		IF conveyorPos >= currentBundle.length AND NOT occupied THEN //rear of bundle has cleared the area
			status := SectionTask.COMPLETE;
		END_IF
		
	SectionTask.COMPLETE:	
		iBundle := iBundle + 1;
		//bundleOut := GVL.nullBundle;
		MEMSET(ADR(activeBundle), 0, SIZEOF(activeBundle));
		
		status := SectionTask.IDLE;
		
		runSectionTasks := TRUE;
		
	-100: //previously completed bundle reversed into this section		
		pConveyorMode := ConveyorMode.FORWARD;
		
		IF NOT occupied AND conveyorPos = 0 THEN
			status := SectionTask.ALIGN;
		END_IF
		
END_CASE
END_METHOD

METHOD shiftIterator : BOOL
//2023-10-24 - array of pointers replaced with iterator for MAIN's queue passed by pointer
iBundle := iBundle - 1;
END_METHOD

METHOD PROTECTED ABSTRACT unload : BOOL
VAR_INPUT
END_VAR
(*
unload, unstage, etc
*)
END_METHOD

END_FUNCTION_BLOCK

// ---- DUTs/Hardware/Conveyors/ConveyorSC.TcPOU
FUNCTION_BLOCK ConveyorSC
VAR_INPUT
	bEnable : BOOL;
END_VAR
VAR_OUTPUT
	trueMode : ConveyorMode;
	requestedMode : ConveyorMode;
	
	error AT %I* : BOOL;
	position AT %I* : REAL;
	velocity AT %I* : REAL;
END_VAR
VAR
	enable AT %Q* : BOOL := TRUE;
	direction AT %Q* : BOOL; //FALSE = forward, TRUE = backward
	pulse AT %Q* : BOOL;
	reset AT %Q* : BOOL;
	
	sensorEntry AT %I* : BOOL := TRUE;
	sensorExit AT %I* : BOOL;
END_VAR
VAR
	//nextConveyor : POINTER TO ConveyorSC;
	//prevConveyor : POINTER TO ConveyorSC;
	
	pulser : TP; //pulses are assumed to be low-high-low
END_VAR
VAR_STAT CONSTANT
	pulseWidth : TIME := T#50MS;
END_VAR
(*
standard slat conveyor - no lifter
compliant with PLCopen motion control
*)

enable := bEnable;

override();

sequence();

METHOD backward : BOOL
VAR_INPUT
END_VAR
END_METHOD

METHOD forward : BOOL
VAR_INPUT
END_VAR
END_METHOD

{attribute 'monitoring' := 'call'}
PROPERTY IsOccupied : BOOL
GET
IsOccupied := sensorExit OR sensorEntry;
END_GET
END_PROPERTY

METHOD join : BOOL
VAR_INPUT
	conveyor : POINTER TO ConveyorSC;
END_VAR
//nextConveyor := conveyor;
//conveyor^.prevConveyor := THIS;
END_METHOD

METHOD PROTECTED override : BOOL
VAR_INPUT
END_VAR
END_METHOD

METHOD reset : BOOL
VAR_INPUT
END_VAR
position := 0;
velocity := velocity; //no change
END_METHOD

METHOD PROTECTED sequence : BOOL
VAR_INPUT
END_VAR
direction := (trueMode = ConveyorMode.BACKWARD); //set direction bit

pulser(IN:= , PT:= pulseWidth, Q=> pulse, ET=> );
pulser.IN := 
	enable AND 
	NOT error AND 
	NOT reset AND 
	(trueMode = ConveyorMode.FORWARD OR trueMode = ConveyorMode.BACKWARD)
	AND pulser.Q; //ends pulse itself
END_METHOD

METHOD setMode : BOOL
VAR_INPUT
	mode : ConveyorMode;
END_VAR
trueMode := mode;
END_METHOD

METHOD setRequest : BOOL
VAR_INPUT
	newRequest : ConveyorMode;
END_VAR
requestedMode := newRequest;
END_METHOD

METHOD target : BOOL
VAR_INPUT
	targetPosition : REAL;
END_VAR
END_METHOD

END_FUNCTION_BLOCK

// ---- DUTs/Hardware/Conveyors/Conveyor.TcPOU
FUNCTION_BLOCK Conveyor
VAR_INPUT
	bEnable : BOOL;
END_VAR
VAR_OUTPUT	
	enable AT %Q* : BOOL;
	direction AT %Q* : BOOL; //FALSE = forward, TRUE = backward
	pulse AT %Q* : BOOL;
	reset AT %Q* : BOOL;
	
	error AT %I* : BOOL;
	sensorEntry AT %I* : BOOL;
	sensorExit AT %I* : BOOL;
	
	//vertical conveyors only
	requestLifter: BOOL;

	lifterEnable AT %Q* : BOOL := TRUE;
	lifterDirection AT %Q* : BOOL; //FALSE = up, TRUE = down
	lifterPulse AT %Q* : BOOL;
	lifterReset AT %Q* : BOOL;
	
	lifterError AT %I* : BOOL;
	extended AT %I* : BOOL;
	retracted AT %I* : BOOL;
END_VAR
VAR_OUTPUT
	position AT %I* : REAL;
	velocity AT %I* : REAL;
END_VAR
VAR
	operation : ConveyorMode;
	request : ConveyorMode;
	
	//pulses are assumed to be low-HIGH-low
	pulser : TP;
	lifterPulser : TP;
	
	hasLifter : BOOL;
END_VAR
VAR_STAT CONSTANT
	pulseWidth : TIME := T#25MS;
END_VAR

pulser(IN:= , PT:= pulseWidth, Q=> pulse, ET=> );

direction := (operation = ConveyorMode.BACKWARD);

pulser.IN := 
	enable AND 
	NOT error AND 
	NOT reset AND 
	(operation = ConveyorMode.FORWARD OR operation = ConveyorMode.BACKWARD);

IF pulser.IN AND NOT pulser.Q THEN
	pulser.IN := FALSE;
END_IF

lifterPulser(IN:= , PT:= pulseWidth, Q=> lifterPulse, ET=> );

lifterPulser.IN := 
	hasLifter AND
	lifterEnable AND 
	NOT lifterError AND 
	NOT lifterReset AND 
	requestLifter;
	
IF lifterPulser.IN AND NOT lifterPulser.Q THEN
	lifterPulser.IN := FALSE;
END_IF

METHOD backward : BOOL
VAR_INPUT
END_VAR
END_METHOD

METHOD extend : BOOL
VAR_INPUT
END_VAR
END_METHOD

METHOD forward : BOOL
VAR_INPUT
END_VAR
END_METHOD

{attribute 'monitoring' := 'call'}
PROPERTY IsOccupied : BOOL
GET
IsOccupied := sensorExit OR sensorEntry;
END_GET
END_PROPERTY

METHOD reset : BOOL
VAR_INPUT
END_VAR
position := 0;
velocity := velocity; //no change

extend();
END_METHOD

METHOD retract : BOOL
VAR_INPUT
END_VAR
END_METHOD

METHOD setOperation : BOOL
VAR_INPUT
	newOperation : ConveyorMode;
END_VAR
operation := newOperation;
END_METHOD

METHOD setRequest : BOOL
VAR_INPUT
	newRequest : ConveyorMode;
END_VAR
request := newRequest;
END_METHOD

METHOD target : BOOL
VAR_INPUT
	targetPosition : REAL;
END_VAR
END_METHOD

END_FUNCTION_BLOCK

// ---- DUTs/Hardware/Robots/RobotA22.TcPOU
FUNCTION_BLOCK RobotA22 EXTENDS KukaRobot
VAR_INPUT
	wrapSafety : BOOL;
END_VAR
VAR_OUTPUT //from outputs array
	taskID : TaskA22;
	param1 : INT;
	param2 : INT;
	Xmm : INT;
	Ymm : INT;
	Zmm : INT;
	angle : INT;
	foldPosition0 : INT;
	foldPosition1 : INT;
END_VAR
VAR_OUTPUT //from inputs array
	tool : SectionEnum := SectionEnum.CARDBOARD_CORNERGUARD;
	suspendedMaterial : STRING;
	
	completedTask : TaskA22;
	eoatDistance : INT;
	cardboardAvailability : INT;
	cornerGuardAvailability : INT;
	materialAtHoldingPosition : INT;
	//grp6
	//grp7
	
	wrapSafetyIn : BOOL;
	
END_VAR
VAR //HMI data
	reservationEnum : SectionEnum;
	hmiTask : STRING;
	hmiTool : STRING;
END_VAR

{warning disable C0195}
SUPER^();

outputs[1] := taskID;
outputs[2] := param1;
outputs[3] := param2;
outputs[4] := Xmm;
outputs[5] := Ymm;
outputs[6] := Zmm;
outputs[7] := angle;
outputs[8] := foldPosition0;
outputs[9] := foldPosition1;

refreshParameters();

reservationEnum := reservation;
IF reservationEnum = SectionEnum.NULL_SECTION THEN
	hmiReservation := 'N/A';
ELSE
	hmiReservation := TO_STRING(reservationEnum);
END_IF

hmiTask := TO_STRING(taskID);
hmiTool := TO_STRING(tool);

{attribute 'monitoring' := 'call'}
PROPERTY Busy : BOOL
GET
VAR
	//emptyOutput : ARRAY[1..50] OF INT;
END_VAR
//Busy stays TRUE until outputs are cleared AND completed task has elapsed
//Ready is always inverse of Busy
refreshParameters();

Busy := taskID <> 0 OR completedTask <> 0;
END_GET
END_PROPERTY

METHOD changeEOAT : BOOL
VAR_INPUT
	targetTool : SectionEnum;
END_VAR
//fill in IO here

changeEOAT := TRUE;
END_METHOD

METHOD clearCommand : BOOL
VAR_INPUT
END_VAR
SUPER^.clearCommand();

refreshParameters();
END_METHOD

{attribute 'monitoring' := 'call'}
PROPERTY Done : BOOL
GET
refreshParameters();

Done :=
	completedTask = taskID AND
	taskID <> 0 AND
	completedTask <> 0;
END_GET
END_PROPERTY

{attribute 'monitoring' := 'call'}
PROPERTY HoldMaterial : STRING
GET
HoldMaterial := suspendedMaterial;
END_GET
SET
suspendedMaterial := HoldMaterial;
END_SET
END_PROPERTY

{attribute 'monitoring' := 'call'}
PROPERTY Ready : BOOL
GET
refreshParameters();

Ready := taskID = 0 AND completedTask = 0;
END_GET
END_PROPERTY

METHOD PRIVATE refreshParameters : BOOL
VAR_INPUT
END_VAR
{warning disable C0196}
taskID := outputs[1];
param1 := outputs[2];
param2 := outputs[3];
Xmm := outputs[4];
Ymm := outputs[5];
Zmm := outputs[6];
angle := outputs[7];
foldPosition0 := outputs[8];
foldPosition1 := outputs[9];

completedTask := inputs[1];
(*
eoatDistance := inputs[2];
magazineAvailability := inputs[3];
chipboardSkidInPosition := inputs[4];
materialAtHoldingPosition := inputs[5];
//robotEOAT := inputs[6];

strapSafetyIn := inputs[4].15;
*)
END_METHOD

METHOD setGroup : BOOL
VAR_INPUT
	group : INT;
	value : INT;
END_VAR
SUPER^.setGroup(group := group, value := value);

refreshParameters();
END_METHOD

METHOD setParameters : BOOL
VAR_INPUT
	newTaskID : INT;
	newParam1 : INT;
	newParam2 : INT;
	newXmm : INT;
	newYmm : INT;
	newZmm : INT;
	newAngle : INT;
	newStagingOccupancy : INT;
	newInsertionSuctionStatus : INT;
	newMagazineStatus : INT; //unused
	newInspectionValue : INT;
END_VAR
setGroup(group := 1, value := newTaskID);
setGroup(group := 2, value := newParam1);
setGroup(group := 3, value := newParam2);
setGroup(group := 4, value := newXmm);
setGroup(group := 5, value := newYmm);
setGroup(group := 6, value := newZmm);
setGroup(group := 7, value := newAngle);

newStagingOccupancy.15 := wrapSafety;
setGroup(group := 8, value := newStagingOccupancy);

setGroup(group := 9, value := newInsertionSuctionStatus);
setGroup(group := 10, value := newMagazineStatus);
setGroup(group := 11, value := newInspectionValue);

refreshParameters();
END_METHOD

END_FUNCTION_BLOCK

// ---- DUTs/Hardware/Material Holders/SkidMagazine.TcPOU
FUNCTION_BLOCK SkidMagazine EXTENDS MaterialHolder
VAR_OUTPUT
	inPosition AT %I* : ARRAY[1..2] OF BOOL;
END_VAR

SUPER^();

METHOD setOccupancy : BOOL
VAR_INPUT
	i : INT;
	occupancy : BOOL;
END_VAR
VAR_OUTPUT
	errorBounds : BOOL;
END_VAR
errorBounds := i < LOWER_BOUND(slots, 1) OR i > UPPER_BOUND(slots, 1);

IF NOT errorBounds THEN
	slots[i].occupied := occupancy;
END_IF
END_METHOD

END_FUNCTION_BLOCK

// ---- DUTs/Hardware/Insertion Package/Insertion.TcPOU
FUNCTION_BLOCK Insertion //2d insertion that combines a slider (alignment) and screw (push)
VAR_INPUT //interface references to existing drives
	slider : I_PositionalDrive;
	screw : I_ContinuousDrive;
END_VAR
VAR_OUTPUT
	contact AT %I* : BOOL;
	
	active : BOOL;
	error : BOOL;
	home : BOOL;
	
	homingComplete : BOOL;
	
	sliderPos : LREAL;
END_VAR
(*
this FB encapsulates 2 drives into a generic insertion machine
both drives should be declared externally in Hardware GVL as a concrete FB
Insertion instance should be declared and called in module scope, with the drives from Hardware GVL passed in by Interface reference
*)

homingComplete := slider.HomeSet AND screw.HomeSet;

active := slider.Active OR screw.Active;
error := slider.Error OR screw.Error;
home := slider.AtHome AND screw.AtHome;

sliderPos := slider.CurrentPosition;

METHOD align : BOOL
VAR_INPUT
	targetPos : REAL;
END_VAR
slider.moveAbsolute(newTarget := targetPos);
END_METHOD

METHOD homingSequence : BOOL
VAR_INPUT
END_VAR
IF NOT slider.homeSet THEN
	slider.homingSequence();
END_IF

IF NOT screw.homeSet THEN
	screw.homingSequence();
END_IF

homingSequence := homingComplete;
END_METHOD

METHOD press : BOOL
VAR_INPUT
END_VAR
IF NOT contact THEN
	screw.moveContinuous(direction := MC_Negative_Direction);
END_IF
END_METHOD

METHOD release : BOOL
VAR_INPUT
END_VAR
screw.moveContinuous(direction := MC_Positive_Direction);
END_METHOD

METHOD reset : BOOL
VAR_INPUT
END_VAR
slider.reset();
screw.reset();
END_METHOD

METHOD stop : BOOL
VAR_INPUT
END_VAR
screw.stop();
slider.stop();
END_METHOD

METHOD toHome : BOOL
VAR_INPUT
END_VAR
slider.toHome();
screw.toHome();

toHome := slider.AtHome AND screw.AtHome;
END_METHOD

END_FUNCTION_BLOCK

// ---- POUs/Helper Functions/Material Functions/MatchesMaterialType.TcPOU
FUNCTION MatchesMaterialType : BOOL
VAR_INPUT
	pair : REFERENCE TO PositionMaterials;
	materialPrefix : STRING;
END_VAR
VAR
END_VAR

MatchesMaterialType :=
	FIND(pair.top, materialPrefix) > 0 AND
	FIND(pair.left, materialPrefix) > 0 AND
	FIND(pair.right, materialPrefix) > 0 AND
	FIND(pair.bottom, materialPrefix) > 0 AND
	
	FIND(pair.topLeft, materialPrefix) > 0 AND
	FIND(pair.topRight, materialPrefix) > 0 AND
	FIND(pair.bottomLeft, materialPrefix) > 0 AND
	FIND(pair.bottomRight, materialPrefix) > 0 ;

END_FUNCTION

// ---- Sections/A21a - Chipboard/ChipboardEx.TcPOU
FUNCTION_BLOCK ChipboardEx EXTENDS SectionEx
VAR_IN_OUT
	A21_SC_C18 : ConveyorSC;
	A21_LSC_C19 : ConveyorLSC;
	A21_LSC_C20 : ConveyorLSC;
END_VAR
VAR_IN_OUT
	robotLeft, robotRight : RobotA21;
	toolStorageLeft, toolStorageRight : A21ToolStorage;
	
	skidLeft, skidRight : SkidMagazine;
END_VAR
VAR	
	step : (IDLE, RETRACT_CONVEYOR, LOAD_CIP, EXTEND_CONVEYOR, COMPLETE := 1050);
	
	loadSet : INT;
END_VAR
VAR //bundle data
	materialsArr : (*REFERENCE TO*) ARRAY[0..CONSTS.maxPairs] OF PositionMaterials;
END_VAR
VAR
	aoiLoadLeft, aoiLoadRight : AOI_LoadChipboard;
	
	pushSmallConveyorPos : REAL;
	pushLargeConveyorPos : REAL;
END_VAR

aoiBlocks(); //call AOIs and large library FBs

SUPER^();

METHOD PROTECTED aoiBlocks : BOOL
VAR_INPUT
END_VAR
{warning disable C0371}
aoiLoadRight(
	sectionID:= sectionID, 
	execute:= ,
	robot:= robotRight, 
	storage:= skidRight,
	loadedMaterials:= loadedMaterials,
	surfaceID:= , 
	material:= , 
	loadedMaterials=> , 
	done=> , 
	error=> );
	
aoiLoadRight(
	sectionID:= sectionID, 
	execute:= , 
	robot:= robotRight, 
	storage:= skidRight,
	loadedMaterials:= loadedMaterials, 
	surfaceID:= , 
	material:= , 
	busy=> , 
	done=> , 
	error=> , 
	recovery=> , 
	failCounter=> );
END_METHOD

METHOD PROTECTED load : BOOL
VAR_INPUT
	pairIndex : INT;
END_VAR
VAR_OUTPUT
	error : BOOL;
END_VAR
VAR
	pair : REFERENCE TO PositionMaterials REF= materialsArr[pairIndex];
END_VAR
{warning disable C0371}
IF robotLeft.error AND robotLeft.error THEN
	error := TRUE;
	RETURN;

ELSIF
	( robotLeft.reservation <> sectionID AND_THEN robotLeft.reserve(sectionID) ) OR
	( robotRight.reservation <> sectionID AND_THEN robotRight.reserve(sectionID) ) THEN
	RETURN;
	
ELSIF //wrong tool and not finished changing tool
	(robotLeft.tool <> sectionID AND_THEN NOT robotLeft.changeEOAT(targetTool := sectionID)) OR
	(robotRight.tool <> sectionID AND_THEN NOT robotRight.changeEOAT(targetTool := sectionID))
THEN
	RETURN;
END_IF
//robots ok

CASE loadSet OF
	0: //left robot -> top, right robot -> bottom
		IF aoiLoadLeft.done AND aoiLoadRight.done THEN
			aoiLoadLeft.execute := aoiLoadRight.execute := FALSE;
			loadSet := 10;
			RETURN;
		END_IF
		
		aoiLoadLeft.surfaceID := Surface.TOP;
		aoiLoadLeft.material := pair.left;
		
		aoiLoadRight.surfaceID := Surface.BOTTOM;
		aoiLoadRight.material := pair.right;
		
		aoiLoadLeft.execute := NOT aoiLoadLeft.recovery;
		aoiLoadRight.execute := NOT aoiLoadRight.recovery;
		
	10: //recovery		
		IF robotRight.error THEN //left ok, right error
			
			IF aoiLoadLeft.done THEN
				aoiLoadLeft.execute := FALSE;
				loadSet := COMPLETE;
				RETURN;
			END_IF
			
			aoiLoadLeft.surfaceID := Surface.BOTTOM;
			aoiLoadLeft.material := pair.bottom;
			aoiLoadLeft.execute := NOT aoiLoadLeft.recovery;
			
		ELSIF robotLeft.error THEN //left error, right ok
			
			IF aoiLoadRight.done THEN
				aoiLoadRight.execute := FALSE;
				loadSet := COMPLETE;
				RETURN;
			END_IF
			
			aoiLoadRight.surfaceID := Surface.TOP;
			aoiLoadRight.material := pair.top;
			aoiLoadRight.execute := NOT aoiLoadRight.recovery;
			
		END_IF
		
	COMPLETE:
		loadSet := 0;
		
		robotLeft.release(sectionID);
		robotRight.release(sectionID);
		
		load := TRUE;
END_CASE
END_METHOD

METHOD PRIVATE loadingSequence : BOOL
VAR_IN_OUT
	robot : RobotA21;
	storage : SkidMagazine;
	loadStep : INT;
END_VAR
VAR_INPUT
	surfaceID : Surface;
	material : STRING;
END_VAR
VAR_OUTPUT
	fail : BOOL;
END_VAR
VAR
	slot : INT;
END_VAR
VAR CONSTANT
	suctionDistance : INT := 10;
END_VAR
{warning disable C0371}
IF material = '' THEN
	loadingSequence := TRUE;
	RETURN;
END_IF

CASE loadStep OF
	0:
		robot.clearCommand();
		IF robot.Ready THEN
			loadStep := 1;
		END_IF
	
	1:
		IF surfaceID = Surface.BOTTOM (*AND_THEN conveyors not retracted*) THEN
			//retract conveyors
			RETURN;
		END_IF
		loadStep := 10;
		
	10: //grab from chipboard skid
		IF NOT storage.findSlot(material := material, index => slot) THEN
			fail := TRUE;
			RETURN;
		(*
		ELSIF surfaceID = Surface.BOTTOM (*AND_THEN (*conveyor not lowered*)*) THEN
			//lower conveyor
			RETURN;
		*)
		END_IF
		
		IF robot.eoatDistance < suctionDistance THEN
			robot.HoldMaterial := storage.getSlot(i := slot);
		END_IF
		
		IF robot.Done THEN
			loadStep := COMPLETE;
			RETURN;
		ELSIF robot.materialAtHoldingPosition.4 OR robot.materialAtHoldingPosition.5 THEN //bits 4 and 5 are chipboard in position
			loadStep := 20;
			RETURN;
		END_IF
		
		robot.setGroup(group := 1, value := TaskA21.PLACE_CHIPBOARD_TOP);
		robot.setGroup(group := 2, value := slot);
		
	20: //place to bundle
		IF robotLeft.Done THEN
			loadStep := COMPLETE;
			RETURN;
		END_IF
		
		IF robot.HoldMaterial <> '' THEN
			loadedMaterials[surfaceID] := robot.HoldMaterial;
			robot.HoldMaterial := '';
		END_IF
		
	COMPLETE:
		IF loadedMaterials[surfaceID] = material THEN
			loadingSequence := TRUE;
		ELSE
			loadStep := 0;
		END_IF
		
END_CASE
END_METHOD

METHOD PROTECTED maintenance : BOOL
VAR_INPUT
END_VAR
{warning disable C0371}
//no specific tasks yet, free run and testing

IF robotLeft.Done THEN
	robotLeft.clearCommand();
END_IF

IF robotRight.Done THEN
	robotRight.clearCommand();
END_IF
END_METHOD

METHOD PROTECTED manual : BOOL
VAR_INPUT
END_VAR
END_METHOD

METHOD PROTECTED process : BOOL
VAR_INPUT
	auto : BOOL;
END_VAR
VAR_OUTPUT
	error : BOOL;
END_VAR
CASE step OF
	IDLE:
		IF trigger.Q THEN
			step := RETRACT_CONVEYOR;
		END_IF
		
	RETRACT_CONVEYOR:
		(*
		IF demoPair.bottom <> '' (*retract conveyors*) THEN
			IF TRUE (*BLSC 1-3 retracted*) THEN
				done := TRUE;
			END_IF
		ELSE
			done := TRUE;
		END_IF
		
		IF
			(manualStep AND_THEN execute) OR
			(NOT manualStep AND_THEN done)
		THEN
			done := FALSE;
			step := LOAD_MATERIAL;
		END_IF
		*)
		step := LOAD_CIP;
	LOAD_CIP:
		IF NOT done THEN
			done := load(pairIndex:= iPair, error=> error);
		END_IF
		
		IF
			(auto AND done) OR
			(NOT auto AND_THEN trigger.Q)
		THEN
			done := FALSE;
			
			step := EXTEND_CONVEYOR;
		END_IF
		
	EXTEND_CONVEYOR:
		(*
		IF FALSE (*conveyors not extended*) THEN
			//extend conveyors
		END_IF
		
		IF
			(auto AND done) OR
			(NOT auto AND_THEN execute) //conveyors extended
		THEN
			done := FALSE;
			step := COMPLETE;
		END_IF
		*)
		step := COMPLETE;
	COMPLETE:
		//reset everything
		step := IDLE;
		
		process := TRUE;
		
END_CASE
END_METHOD

METHOD PROTECTED ps_AbortCondition : BOOL
VAR_INPUT
END_VAR
{warning disable C0371}
ps_AbortCondition :=
	robotLeft.error OR 
	robotRight.error;
END_METHOD

METHOD PROTECTED ps_Aborted : BOOL
VAR_INPUT
END_VAR
ps_Aborted := TRUE;
END_METHOD

METHOD PROTECTED ps_Aborting : BOOL
VAR_INPUT
END_VAR
{warning disable C0371}
aoiLoadLeft.reset();
aoiLoadRight.reset();

robotLeft.clearCommand();
robotRight.clearCommand();

//stop conveyors

ps_Aborting :=
	NOT robotLeft.Busy AND
	NOT robotRight.Busy;
END_METHOD

METHOD PROTECTED ps_Clearing : BOOL
VAR_INPUT
END_VAR
{warning disable C0371}
(*reset conveyors*)

ps_Clearing := 
	NOT robotLeft.error AND
	NOT robotRight.error;
END_METHOD

METHOD PROTECTED ps_Complete : BOOL
VAR_INPUT
END_VAR
ps_Complete := TRUE;
END_METHOD

METHOD PROTECTED ps_Completing : BOOL
VAR_INPUT
END_VAR
ps_Completing := NOT occupied;
END_METHOD

METHOD PROTECTED ps_Held : BOOL
VAR_INPUT
END_VAR
ps_Held := NOT hold;
END_METHOD

METHOD PROTECTED ps_HoldCondition : BOOL
VAR_INPUT
END_VAR
END_METHOD

METHOD PROTECTED ps_Holding : BOOL
VAR_INPUT
END_VAR
{warning disable C0371}
//set robot to pause

ps_Holding := TRUE;
END_METHOD

METHOD PROTECTED ps_Resetting : BOOL
VAR_INPUT
END_VAR
{warning disable C0371}
(*reset conveyors*)

ps_Resetting := 
	reset AND
	NOT robotLeft.error AND
	NOT robotRight.error;
END_METHOD

METHOD PROTECTED ps_Starting : BOOL
VAR_INPUT
END_VAR
{warning disable C0371}
//extend conveyors

ps_Starting := TRUE; //conveyors extended
END_METHOD

METHOD PROTECTED ps_StopCondition : BOOL
VAR_INPUT
END_VAR
ps_StopCondition := 
	stop;
END_METHOD

METHOD PROTECTED ps_Stopped : BOOL
VAR_INPUT
END_VAR
ps_Stopped := TRUE;
END_METHOD

METHOD PROTECTED ps_Stopping : BOOL
VAR_INPUT
END_VAR
{warning disable C0371}
aoiLoadLeft.reset();
aoiLoadRight.reset();

robotLeft.clearCommand();
robotRight.clearCommand();

//stop conveyors

ps_Stopping :=
	NOT robotLeft.Busy AND
	NOT robotRight.Busy;
END_METHOD

METHOD PROTECTED ps_SuspendCondition : BOOL
VAR_INPUT
END_VAR
END_METHOD

METHOD PROTECTED ps_Suspended : BOOL
VAR_INPUT
END_VAR
ps_Suspended := NOT ps_SuspendCondition();
END_METHOD

METHOD PROTECTED ps_Suspending : BOOL
VAR_INPUT
END_VAR
ps_Suspending := TRUE;
END_METHOD

METHOD PROTECTED ps_Unholding : BOOL
VAR_INPUT
END_VAR
ps_Unholding := TRUE;
END_METHOD

METHOD PROTECTED ps_Unsuspending : BOOL
VAR_INPUT
END_VAR
ps_Unsuspending := TRUE;
END_METHOD

METHOD PROTECTED runSectionTasks : BOOL
VAR_INPUT
	auto : BOOL;
END_VAR
VAR_OUTPUT
	error : BOOL;
END_VAR
SUPER^.runSectionTasks(auto := auto, error => error);

CASE status OF //add additional instructions for each state
	SectionTask.IDLE:
		//
	
	SectionTask.ALIGN:
		//
		
	SectionTask.ACTIVE:
		//
		
	SectionTask.DISCHARGE:
		aoiLoadLeft.reset();
		aoiLoadRight.reset();
		
	SectionTask.COMPLETE:	
		//
		
	-100:
		RETURN;
		
END_CASE
END_METHOD

METHOD PROTECTED unload : BOOL
VAR_INPUT
END_VAR
//unload from insertion
//remove from staging table
END_METHOD

END_FUNCTION_BLOCK

// ---- DUTs/Hardware/Robots/RobotA21.TcPOU
FUNCTION_BLOCK RobotA21 EXTENDS KukaRobot
VAR_INPUT
	strapSafety : BOOL;
END_VAR
VAR_OUTPUT //from outputs array
	{warning disable C0195}
	taskID : TaskA21;
	param1 : INT;
	param2 : INT;
	Xmm : INT;
	Ymm : INT;
	Zmm : INT;
	angle : INT;
	stagingOccupancy : INT;
	insertionSuctionStatus : INT;
	magazineStatus : INT; //unused
	inspectionValue : INT;
	
	strapSafetyOut : BOOL;
END_VAR
VAR_OUTPUT //from inputs array
	tool : SectionEnum := SectionEnum.WOOD_BUNK;
	suspendedMaterial : STRING;
	
	completedTask : TaskA21;
	eoatDistance : INT;
	woodBunkAvailability : INT;
	chipboardAvailability : INT;
	materialAtHoldingPosition : INT;
	
	strapSafetyIn : BOOL;
END_VAR
VAR
	reservationEnum : SectionEnum;
	hmiTask : STRING;
	hmiTool : STRING;
END_VAR
(*
extends KukaRobot
	assigns descriptive labels to each IO group from the array
	additional section-specific methods to get/set IO groups
*)

(*
parameters - aliases to IO elements
command - full IO array
*)
{warning disable C0195}
SUPER^();

outputs[1] := taskID;
outputs[2] := param1;
outputs[3] := param2;
outputs[4] := Xmm;
outputs[5] := Ymm;
outputs[6] := Zmm;
outputs[7] := angle;
outputs[8] := stagingOccupancy;
outputs[9] := insertionSuctionStatus;
outputs[10] := magazineStatus;
outputs[11] := inspectionValue;

outputs[8].15 := strapSafety;

refreshParameters();

reservationEnum := reservation;
IF reservationEnum = SectionEnum.NULL_SECTION THEN
	hmiReservation := 'N/A';
ELSE
	hmiReservation := TO_STRING(reservationEnum);
END_IF

hmiTask := TO_STRING(taskID);
hmiTool := TO_STRING(tool);

{attribute 'monitoring' := 'call'}
PROPERTY Busy : BOOL
GET
VAR
	//emptyOutput : ARRAY[1..50] OF INT;
END_VAR
//Busy stays TRUE until outputs are cleared AND completed task has elapsed
//Ready is always inverse of Busy
refreshParameters();

Busy := taskID <> 0 OR completedTask <> 0;
END_GET
END_PROPERTY

METHOD changeEOAT : BOOL
VAR_INPUT
	targetTool : SectionEnum;
END_VAR
setGroup(group := 1, value := TaskA21.TOOL_CHANGE_CHIPBOARD);
setGroup(group := 1, value := TaskA21.TOOL_CHANGE_BUNK);

changeEOAT := tool = targetTool;
END_METHOD

METHOD clearCommand : BOOL
VAR_INPUT
END_VAR
SUPER^.clearCommand();

refreshParameters();
END_METHOD

{attribute 'monitoring' := 'call'}
PROPERTY Done : BOOL
GET
refreshParameters();

Done :=
	completedTask = taskID AND
	taskID <> 0 AND
	completedTask <> 0;
END_GET
END_PROPERTY

{attribute 'monitoring' := 'call'}
PROPERTY HoldMaterial : STRING
GET
HoldMaterial := suspendedMaterial;
END_GET
SET
suspendedMaterial := HoldMaterial;
END_SET
END_PROPERTY

{attribute 'monitoring' := 'call'}
PROPERTY Ready : BOOL
GET
refreshParameters();

Ready := taskID = 0 AND completedTask = 0;
END_GET
END_PROPERTY

METHOD PRIVATE refreshParameters : BOOL
VAR_INPUT
END_VAR
{warning disable C0196}
taskID := outputs[1];
param1 := outputs[2];
param2 := outputs[3];
Xmm := outputs[4];
Ymm := outputs[5];
Zmm := outputs[6];
angle := outputs[7];
stagingOccupancy := outputs[8];
insertionSuctionStatus := outputs[9];
magazineStatus := outputs[10]; //unused
inspectionValue := outputs[11];

completedTask := inputs[1];
eoatDistance := inputs[2];
woodBunkAvailability := inputs[3];
chipboardAvailability := inputs[4];
materialAtHoldingPosition := inputs[5];
//robotEOAT := inputs[6];

strapSafetyIn := inputs[4].15;
END_METHOD

METHOD setGroup : BOOL
VAR_INPUT
	group : INT;
	value : INT;
END_VAR
SUPER^.setGroup(group := group, value := value);

refreshParameters();
END_METHOD

METHOD setParameters : BOOL
VAR_INPUT
	newTaskID : INT;
	newParam1 : INT;
	newParam2 : INT;
	newXmm : INT;
	newYmm : INT;
	newZmm : INT;
	newAngle : INT;
	newStagingOccupancy : INT;
	newInsertionSuctionStatus : INT;
	newMagazineStatus : INT; //unused
	newInspectionValue : INT;
END_VAR
VAR_INPUT
	strapSafety : BOOL;
END_VAR
setGroup(group := 1, value := newTaskID);
setGroup(group := 2, value := newParam1);
setGroup(group := 3, value := newParam2);
setGroup(group := 4, value := newXmm);
setGroup(group := 5, value := newYmm);
setGroup(group := 6, value := newZmm);
setGroup(group := 7, value := newAngle);

newStagingOccupancy.15 := strapSafety;
setGroup(group := 8, value := newStagingOccupancy);

setGroup(group := 9, value := newInsertionSuctionStatus);
setGroup(group := 10, value := newMagazineStatus);
setGroup(group := 11, value := newInspectionValue);

refreshParameters();
END_METHOD

END_FUNCTION_BLOCK

// ---- Sections/A21b - Wood Bunk/WoodBunkEx.TcPOU
FUNCTION_BLOCK WoodBunkEx EXTENDS SectionEx
VAR_IN_OUT
	A21_LSC_C21 : ConveyorLSC;
END_VAR
VAR_IN_OUT
	robotLeft, robotRight : RobotA21;
	toolStorageLeft, toolStorageRight : A21ToolStorage;
	
	stagingTableLeft, stagingTableRight : StagingTable;
	magazineLeft, magazineRight : SkidMagazine;
	
	strapper : StrapMachine;
	
	insertionLeft, insertionRight : Insertion;
	pistonBottom : SimplePiston;
	
	suctionTop : ARRAY[*] OF SuctionPad; (*1..3*)
	suctionLeft : ARRAY[*] OF SuctionPad; (*1..4*)
	suctionRight : ARRAY[*] OF SuctionPad; (*1..4*)
	suctionBottom : ARRAY[*] OF SuctionPad; (*1..2*)
END_VAR
VAR
	step : (IDLE, STAGING, LOAD_WB, PUSH, STRAP, RELEASE, COMPLETE := 1050);
	
	stageStepLeft, stageStepRight : INT;
	loadStepLeft, loadStepRight : INT;
END_VAR
VAR //bundle data
	demoHeight : REAL := 640; //mm
	materialsArr : (*REFERENCE TO*) ARRAY[0..CONSTS.maxPairs] OF PositionMaterials;
END_VAR
VAR
	//AOIs encapsulate functionality and reduce the number of module variables
	aoiTemplateLeft, aoiTemplateRight : AOI_StagingTemplate;
	aoiStageLeft, aoiStageRight : AOI_StageWoodBunk; 
	aoiLoadLeft, aoiLoadRight : AOI_LoadWoodBunk;
	
	suctionRelease : TON;
	
	//for testing, to be removed when deployoed
	latchLeft, latchRight : BOOL; //prevents SMC sliders from overshooting
	suctionEnableTop, suctionEnableLeft, suctionEnableRight, suctionEnableBottom : BOOL;
END_VAR

conveyorPos := A21_LSC_C21.position;

aoiBlocks();

SUPER^();

(*
any PackML state-methods that SectionEx has a concrete implementation for will be overriden by concrete FBs that extend it
(ie: all or most of them)

to call the base implementation, add:
	SUPER^.ps_<state>();
to the concrete FB's implementation of that state-method
*)

METHOD PROTECTED aoiBlocks : BOOL
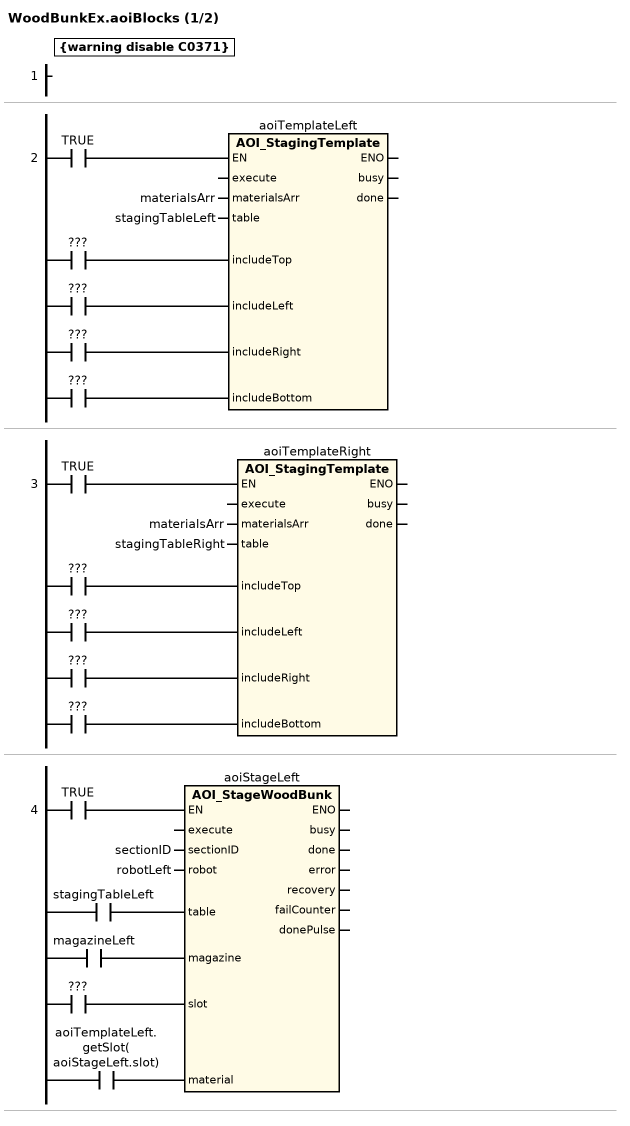
// NETWORK 1
// label: {warning disable C0371}

// NETWORK 2
aoiTemplateLeft(materialsArr := materialsArr, table := stagingTableLeft); // AOI_StagingTemplate

// NETWORK 3
aoiTemplateRight(materialsArr := materialsArr, table := stagingTableRight); // AOI_StagingTemplate

// NETWORK 4
aoiStageLeft(
    sectionID := sectionID,
    robot := robotLeft,
    table := stagingTableLeft,
    magazine := magazineLeft,
    material := aoiTemplateLeft.getSlot(aoiStageLeft.slot)); // AOI_StageWoodBunk

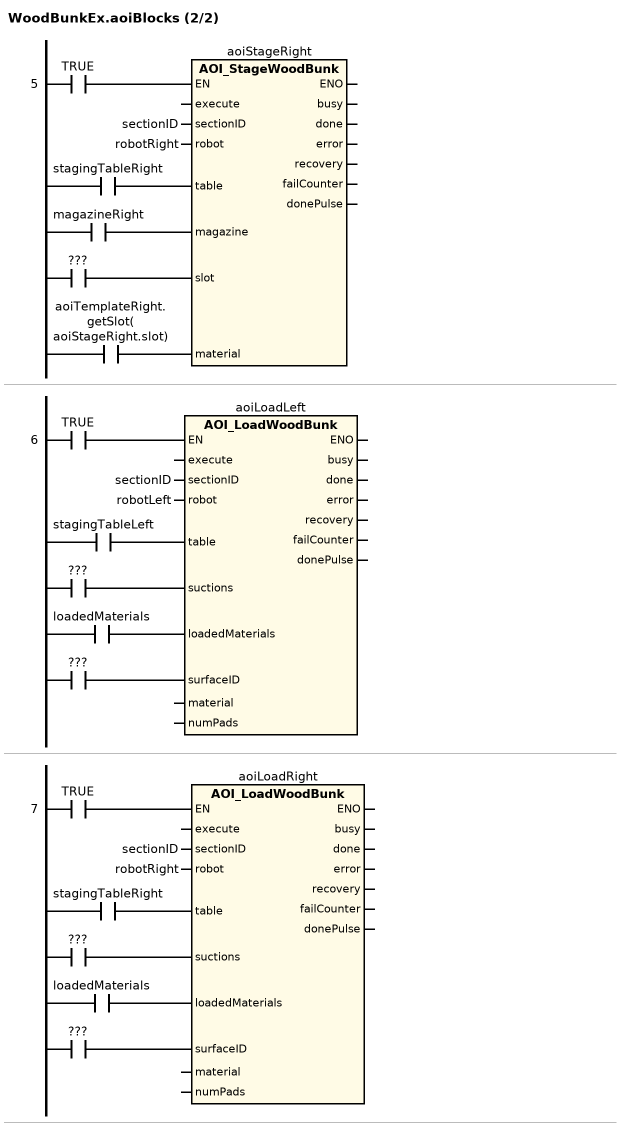
// NETWORK 5
aoiStageRight(
    sectionID := sectionID,
    robot := robotRight,
    table := stagingTableRight,
    magazine := magazineRight,
    material := aoiTemplateRight.getSlot(aoiStageRight.slot)); // AOI_StageWoodBunk

// NETWORK 6
aoiLoadLeft(
    sectionID := sectionID,
    robot := robotLeft,
    table := stagingTableLeft,
    loadedMaterials := loadedMaterials); // AOI_LoadWoodBunk

// NETWORK 7
aoiLoadRight(
    sectionID := sectionID,
    robot := robotRight,
    table := stagingTableRight,
    loadedMaterials := loadedMaterials); // AOI_LoadWoodBunk
END_METHOD

METHOD PROTECTED load : BOOL
VAR_INPUT
	pairIndex : INT;
END_VAR
VAR_OUTPUT
	error : BOOL;
END_VAR
VAR
	pair : REFERENCE TO PositionMaterials REF= materialsArr[pairIndex];
	errorLeft, errorRight : BOOL;
END_VAR
{warning disable C0371}
(*
loading sequences are independent as each side has its own step variable
can be extended by changing the include<> parameters
*)

load :=
	loadEx(
		robot:= robotLeft, 
		aoiLoad:= aoiLoadLeft, 
		loadStep:= loadStepLeft, 
		pairIndex:= pairIndex, 
		includeTop:= TRUE, 
		includeLeft:= TRUE, 
		includeRight:= FALSE, 
		includeBottom:= FALSE, 
		error=> errorLeft)
	AND
	loadEx(
		robot:= robotRight, 
		aoiLoad:= aoiLoadRight, 
		loadStep:= loadStepRight, 
		pairIndex:= pairIndex, 
		includeTop:= FALSE, 
		includeLeft:= FALSE, 
		includeRight:= TRUE, 
		includeBottom:= TRUE, 
		error=> errorRight);
		
error := errorLeft OR errorRight;
END_METHOD

METHOD PRIVATE loadEx : BOOL
VAR_IN_OUT
	robot : RobotA21;
	aoiLoad : AOI_LoadWoodBunk;
	loadStep : INT;
END_VAR
VAR_INPUT
	pairIndex : INT;
	includeTop, includeLeft, includeRight, includeBottom : BOOL;
END_VAR
VAR_OUTPUT
	error : BOOL;
END_VAR
VAR
	pair : REFERENCE TO PositionMaterials REF= materialsArr[pairIndex];
END_VAR
{warning disable C0371}
IF robot.error THEN
	error := TRUE;
	RETURN;
ELSIF robot.reservation <> sectionID AND_THEN NOT robot.reserve(sectionID) THEN
	RETURN;
ELSIF robot.tool <> sectionID AND_THEN NOT robot.changeEOAT(targetTool := sectionID) THEN
	RETURN;
END_IF

error := aoiLoad.error;

CASE loadStep OF
	0:
		loadStep := Surface.TOP;
	
	Surface.TOP:		
		IF NOT includeTop OR aoiLoad.donePulse THEN
			aoiLoad.execute := FALSE;
			aoiLoad.material := '';
			loadStep := Surface.BOTTOM;
			RETURN;
		END_IF
		
		aoiLoad.surfaceID := Surface.TOP;
		aoiLoad.material := pair.top;
		aoiLoad.suctions := suctionTop;
		aoiLoad.numPads := UPPER_BOUND(suctionTop, 1) - LOWER_BOUND(suctionTop, 1) + 1;
		
		aoiLoad.execute := NOT aoiLoad.busy;
		
	Surface.BOTTOM:
		IF NOT includeBottom OR aoiLoad.donePulse THEN
			aoiLoad.execute := FALSE;
			aoiLoad.material := '';
			loadStep := Surface.LEFT;
			RETURN;
		END_IF
		
		aoiLoad.surfaceID := Surface.BOTTOM;
		aoiLoad.material := pair.bottom;
		aoiLoad.suctions := suctionBottom;
		aoiLoad.numPads := UPPER_BOUND(suctionBottom, 1) - LOWER_BOUND(suctionBottom, 1) + 1;
		
		aoiLoad.execute := NOT aoiLoad.busy;
		
	Surface.LEFT:
		IF NOT includeLeft OR aoiLoad.donePulse THEN
			aoiLoad.execute := FALSE;
			aoiLoad.material := '';
			loadStep := Surface.RIGHT;
			RETURN;
		END_IF
		
		aoiLoad.surfaceID := Surface.LEFT;
		aoiLoad.material := pair.left;
		aoiLoad.suctions := suctionLeft;
		aoiLoad.numPads := UPPER_BOUND(suctionLeft, 1) - LOWER_BOUND(suctionLeft, 1) + 1;
		
		aoiLoad.execute := NOT aoiLoad.busy;
		
	Surface.RIGHT:
		IF NOT includeRight OR aoiLoad.donePulse THEN
			aoiLoad.execute := FALSE;
			aoiLoad.material := '';
			loadStep := COMPLETE;
			RETURN;
		END_IF
		
		aoiLoad.surfaceID := Surface.RIGHT;
		aoiLoad.material := pair.right;
		aoiLoad.suctions := suctionRight;
		aoiLoad.numPads := UPPER_BOUND(suctionRight, 1) - LOWER_BOUND(suctionRight, 1) + 1;
		
		aoiLoad.execute := NOT aoiLoad.busy;
		
	COMPLETE:				
		robot.release(sectionID);
		
		aoiLoad.material := '';
		aoiLoad.execute := FALSE;
		
		loadEx := TRUE;
END_CASE
END_METHOD

METHOD PROTECTED maintenance : BOOL
VAR_INPUT
END_VAR
{warning disable C0371}
//no specific tasks yet, free run and testing
SetSuctions(suctionTop, suctionEnableTop);
SetSuctions(suctionLeft, suctionEnableLeft);
SetSuctions(suctionRight, suctionEnableRight);
SetSuctions(suctionBottom, suctionEnableBottom);

IF robotLeft.Done THEN
	robotLeft.clearCommand();
END_IF

IF robotRight.Done THEN
	robotRight.clearCommand();
END_IF
END_METHOD

METHOD PROTECTED manual : BOOL
VAR_INPUT
END_VAR
END_METHOD

METHOD PROTECTED process : BOOL
VAR_INPUT
	auto : BOOL;
END_VAR
VAR_OUTPUT
	error : BOOL;
END_VAR
VAR
	currentPair : REFERENCE TO PositionMaterials REF= materialsArr[iPair];
END_VAR
{warning disable C0371}
IF iPair >= CONSTS.maxPairs THEN
	process := TRUE;
	RETURN;
ELSIF NOT PositionIsValid(pair := currentPair) THEN
	iPair := iPair + 1;
	RETURN;
END_IF

CASE step OF
	IDLE:
		IF auto OR_ELSE trigger.Q THEN
			step := STAGING;
		END_IF

	LOAD_WB:
		IF
			directionCheckAndSet(conveyorPos, currentPair.position) AND 
			( (auto AND done) OR_ELSE (NOT auto AND trigger.Q) )
		THEN
			robotLeft.clearCommand();
			robotRight.clearCommand();
			
			aoiLoadLeft.reset();
			aoiLoadRight.reset();
			
			loadStepLeft := loadStepRight := 0;
			stageStepLeft := stageStepRight := 0;
			
			done := FALSE;
			suctionEnableTop := suctionEnableLeft := suctionEnableRight := suctionEnableBottom := FALSE;
			
			step := PUSH;
			RETURN;
		END_IF
		
		IF NOT done THEN
			done := load(pairIndex := iPair, error => error);
		END_IF
		
		IF NOT auto THEN
			SetSuctions(suctionTop, suctionEnableTop);
			SetSuctions(suctionLeft, suctionEnableLeft);
			SetSuctions(suctionRight, suctionEnableRight);
			SetSuctions(suctionBottom, suctionEnableBottom);
		END_IF
		
	PUSH:
		IF
			(auto AND insertionLeft.contact AND insertionRight.contact AND pistonBottom.extended) OR_ELSE
			(NOT auto AND trigger.Q)
		THEN
			insertionLeft.stop();
			insertionRight.stop();
			
			step := STRAP;
			RETURN;
		END_IF
		
		IF NOT validateInsertion(checkTop:= FALSE, checkLeft:= FALSE, checkRight:= FALSE, checkBottom:= FALSE) THEN
			error := TRUE;
			RETURN;
		END_IF
		
		IF 
			insertionLeft.sliderPos <> demoHeight/2 OR 
			insertionRight.sliderPos <> demoHeight/2
		THEN
			insertionLeft.align(demoHeight/2);
			insertionRight.align(demoHeight/2);
			RETURN;
		END_IF
		
		pistonBottom.extend();
		insertionLeft.press();
		insertionRight.press();
		
	STRAP:
		suctionRelease(IN:= , PT:= suctionReleaseDelay, Q=> , ET=> );
		
		strapper.bEnable := TRUE;
		IF strapper.done THEN
			suctionRelease.IN := FALSE;
			step := RELEASE;
			RETURN;
		END_IF
		
		IF suctionRelease.Q THEN
			SetSuctions(suctionTop, FALSE);
			SetSuctions(suctionLeft, FALSE);
			SetSuctions(suctionRight, FALSE);
			SetSuctions(suctionBottom, FALSE);
		ELSIF strapper.atBundleLevel THEN
			suctionRelease.IN := TRUE;
		END_IF
		
		IF strapper.ready THEN
			strapper.strap();
		END_IF
		
		IF trigger.Q THEN
			suctionRelease.IN := FALSE;
			step := RELEASE;
		END_IF
		
	RELEASE: //release command		
		insertionLeft.toHome();
		insertionRight.toHome();
		pistonBottom.retract();
		
		IF 
			(insertionLeft.screw.AtHome AND insertionRight.screw.AtHome AND pistonBottom.retracted) OR
			trigger.Q
		THEN
			step := COMPLETE;
		END_IF
	
	COMPLETE:
		//reset everything
		iPair := iPair + 1;
		step := IDLE;
END_CASE
END_METHOD

METHOD PROTECTED ps_AbortCondition : BOOL
VAR_INPUT
END_VAR
{warning disable C0371}
ps_AbortCondition :=
	insertionLeft.error OR 
	insertionRight.error OR 
	robotLeft.error OR 
	robotRight.error OR
	strapper.error;
END_METHOD

METHOD PROTECTED ps_Aborted : BOOL
VAR_INPUT
END_VAR
ps_Aborted := TRUE;
END_METHOD

METHOD PROTECTED ps_Aborting : BOOL
VAR_INPUT
END_VAR
{warning disable C0371}
insertionLeft.stop();
insertionRight.stop();
pistonBottom.stop();

aoiLoadLeft.reset();
aoiLoadRight.reset();

aoiStageLeft.reset();
aoiStageRight.reset();

robotLeft.clearCommand();
robotRight.clearCommand();

//stop conveyors

ps_Aborting :=
	NOT insertionLeft.active AND
	NOT insertionRight.active AND
	NOT pistonBottom.busy AND
	NOT robotLeft.Busy AND
	NOT robotRight.Busy;
END_METHOD

METHOD PROTECTED ps_Clearing : BOOL
VAR_INPUT
END_VAR
{warning disable C0371}
insertionLeft.reset();
insertionRight.reset();

ps_Clearing := 
	NOT insertionLeft.error AND
	NOT insertionRight.error AND
	NOT strapper.error AND
	NOT robotLeft.error AND
	NOT robotRight.error;
END_METHOD

METHOD PROTECTED ps_Complete : BOOL
VAR_INPUT
END_VAR
ps_Complete := TRUE;
END_METHOD

METHOD PROTECTED ps_Completing : BOOL
VAR_INPUT
END_VAR
ps_Completing := NOT occupied;
END_METHOD

METHOD PROTECTED ps_Held : BOOL
VAR_INPUT
END_VAR
ps_Held := NOT hold;
END_METHOD

METHOD PROTECTED ps_HoldCondition : BOOL
VAR_INPUT
END_VAR
END_METHOD

METHOD PROTECTED ps_Holding : BOOL
VAR_INPUT
END_VAR
{warning disable C0371}
insertionLeft.stop();
insertionRight.stop();
pistonBottom.stop();
//set robot to pause

ps_Holding :=
	NOT insertionLeft.active AND
	NOT insertionRight.active;
END_METHOD

METHOD PROTECTED ps_Resetting : BOOL
VAR_INPUT
END_VAR
{warning disable C0371}
insertionLeft.reset();
insertionRight.reset();

ps_Resetting := 
	reset AND
	NOT insertionLeft.error AND
	NOT insertionRight.error AND
	NOT strapper.error AND
	NOT robotLeft.error AND
	NOT robotRight.error;
END_METHOD

METHOD PROTECTED ps_Starting : BOOL
VAR_INPUT
END_VAR
{warning disable C0371}
robotLeft.clearCommand();
robotRight.clearCommand();

insertionLeft.homingSequence();
insertionRight.homingSequence();
pistonBottom.retract();

ps_Starting := 
	insertionLeft.screw.HomeSet AND 
	insertionRight.screw.HomeSet AND 
	pistonBottom.retracted;
END_METHOD

METHOD PROTECTED ps_StopCondition : BOOL
VAR_INPUT
END_VAR
ps_StopCondition := 
	stop;
END_METHOD

METHOD PROTECTED ps_Stopped : BOOL
VAR_INPUT
END_VAR
ps_Stopped := TRUE;
END_METHOD

METHOD PROTECTED ps_Stopping : BOOL
VAR_INPUT
END_VAR
{warning disable C0371}
insertionLeft.stop();
insertionRight.stop();
pistonBottom.stop();

aoiLoadLeft.reset();
aoiLoadRight.reset();

aoiStageLeft.reset();
aoiStageRight.reset();

robotLeft.clearCommand();
robotRight.clearCommand();

//stop conveyors

ps_Stopping :=
	NOT insertionLeft.active AND
	NOT insertionRight.active AND
	NOT pistonBottom.busy AND
	NOT robotLeft.Busy AND
	NOT robotRight.Busy;
END_METHOD

METHOD PROTECTED ps_SuspendCondition : BOOL
VAR_INPUT
END_VAR
END_METHOD

METHOD PROTECTED ps_Suspended : BOOL
VAR_INPUT
END_VAR
ps_Suspended := NOT ps_SuspendCondition();
END_METHOD

METHOD PROTECTED ps_Suspending : BOOL
VAR_INPUT
END_VAR
ps_Suspending := TRUE;
END_METHOD

METHOD PROTECTED ps_Unholding : BOOL
VAR_INPUT
END_VAR
ps_Unholding := TRUE;
END_METHOD

METHOD PROTECTED ps_Unsuspending : BOOL
VAR_INPUT
END_VAR
ps_Unsuspending := TRUE;
END_METHOD

METHOD PROTECTED runSectionTasks : BOOL
VAR_INPUT
	auto : BOOL;
END_VAR
VAR_OUTPUT
	error : BOOL;
END_VAR
SUPER^.runSectionTasks(auto := auto, error => error); //basic implementation

CASE status OF //add additional instructions for each status
	SectionTask.IDLE:
		//
	
	SectionTask.ALIGN:
		stage(error => error);
		
	SectionTask.ACTIVE:
		//
		
	SectionTask.DISCHARGE:
		aoiLoadLeft.reset();
		aoiLoadRight.reset();
		
		aoiStageLeft.reset();
		aoiStageRight.reset();
		
		aoiTemplateLeft.reset();
		aoiTemplateRight.reset();
		
	SectionTask.COMPLETE:	
		//
		
	-100:
		//
		
END_CASE
END_METHOD

METHOD PROTECTED stage : BOOL
VAR_OUTPUT
	error : BOOL;
END_VAR
{warning disable C0371}

(*
this method only exists to call stageEx() for both robots
*)
(*
stage := leftDone AND rightDone;

IF NOT leftDone THEN
	leftDone := stageEx(
		robot:= robotLeft, 
		aoiTemplate:= aoiTemplateLeft, 
		aoiStaging:= aoiStageLeft, 
		stageStep:= stageStepLeft, 
		//iSlot:= iSlotLeft, 
		includeTop:= TRUE, 
		includeLeft:= TRUE, 
		includeRight:= FALSE, 
		includeBottom:= FALSE, 
		error=> );
END_IF

IF NOT rightDone THEN
	rightDone := stageEx(
		robot:= robotRight, 
		aoiTemplate:= aoiTemplateRight, 
		aoiStaging:= aoiStageRight, 
		stageStep:= stageStepRight, 
		//iSlot:= iSlotRight, 
		includeTop:= FALSE, 
		includeLeft:= FALSE, 
		includeRight:= TRUE, 
		includeBottom:= TRUE, 
		error=> );
END_IF
*)

stage := 
	stageEx(
		robot:= robotLeft, 
		aoiTemplate:= aoiTemplateLeft, 
		aoiStaging:= aoiStageLeft, 
		stageStep:= stageStepLeft, 
		includeTop:= TRUE, 
		includeLeft:= TRUE, 
		includeRight:= FALSE, 
		includeBottom:= FALSE, 
		error=> )
	AND
	stageEx(
		robot:= robotRight, 
		aoiTemplate:= aoiTemplateRight, 
		aoiStaging:= aoiStageRight, 
		stageStep:= stageStepRight, 
		includeTop:= FALSE, 
		includeLeft:= FALSE, 
		includeRight:= TRUE, 
		includeBottom:= TRUE, 
		error=> );
END_METHOD

METHOD PRIVATE stageEx : BOOL
VAR_IN_OUT
	robot : RobotA21;
	aoiTemplate : AOI_StagingTemplate;
	aoiStaging : AOI_StageWoodBunk;
	stageStep : INT;
END_VAR
VAR_INPUT
	includeTop, includeLeft, includeRight, includeBottom : BOOL;
END_VAR
VAR_OUTPUT
	error : BOOL;
END_VAR
{warning disable C0371}
IF robot.error THEN
	error := TRUE;
	RETURN;
ELSIF robot.reservation <> sectionID AND_THEN NOT robot.reserve(sectionID) THEN
	RETURN;
ELSIF robot.tool <> sectionID AND_THEN NOT robot.changeEOAT(targetTool := sectionID) THEN
	RETURN;
END_IF

CASE stageStep OF
	0: //generate staging template
		IF aoiTemplate.done THEN
			aoiTemplate.execute := FALSE;
			stageStep := 10;
			RETURN;
		END_IF
		
		aoiTemplate.execute := NOT aoiTemplate.busy;
		
		aoiTemplate.includeTop := includeTop;
		aoiTemplate.includeLeft := includeLeft;
		aoiTemplate.includeRight := includeRight;
		aoiTemplate.includeBottom := includeBottom;
		
	10: //stage tables
		IF aoiStaging.slot > 10 THEN
			aoiStaging.execute := FALSE;			
			stageStep := COMPLETE;
			RETURN;
		END_IF
		
		aoiStaging.execute := NOT aoiStaging.busy; //execute if aoiStaging is ready
		
		aoiStaging.slot := MAX(1, aoiStaging.slot); //if 0, sets to 1
		aoiStaging.slot := MIN(aoiStaging.slot, 999); //prevents overflow 
		
		IF aoiStaging.donePulse THEN
			aoiStaging.slot := aoiStaging.slot + 1;
		END_IF
	
	COMPLETE:
		aoiTemplate.clearTemplate();
		aoiTemplate.execute := FALSE;
		aoiStaging.execute := FALSE;
		aoiStaging.reset();
		
		robot.release(sectionID);
		
		aoiStaging.slot := 0;
		
		stageEx := TRUE;
		//stageStep := 0;
END_CASE

error := aoiStaging.error;
END_METHOD

METHOD PROTECTED unload : BOOL
VAR_INPUT
END_VAR
//unload from insertion
//remove from staging table
END_METHOD

METHOD PROTECTED validateInsertion : BOOL
VAR_INPUT
	checkTop : BOOL;
	checkLeft : BOOL;
	checkRight : BOOL;
	checkBottom : BOOL;
END_VAR
validateInsertion := 
	(NOT checkTop OR_ELSE SuctionQuality(suctions:= suctionTop)) AND
	(NOT checkLeft OR_ELSE SuctionQuality(suctions:= suctionLeft)) AND
	(NOT checkRight OR_ELSE SuctionQuality(suctions:= suctionRight)) AND
	(NOT checkBottom OR_ELSE SuctionQuality(suctions:= suctionBottom));

(*
validateSuctionQuality := 
	(
		NOT checkTop OR_ELSE InsertionQuality(
			suctions:= suctionTop, 
			insertionMaterial:= loadedMaterials[Surface.TOP], 
			recipeMaterial:= materialsArr[iPair].top)
	) AND
	(
		NOT checkLeft OR_ELSE InsertionQuality(
			suctions:= suctionLeft, 
			insertionMaterial:= loadedMaterials[Surface.LEFT], 
			recipeMaterial:= materialsArr[iPair].left)
	) AND
	(
		NOT checkRight OR_ELSE InsertionQuality(
			suctions:= suctionRight, 
			insertionMaterial:= loadedMaterials[Surface.RIGHT], 
			recipeMaterial:= materialsArr[iPair].right)
	) AND
	(
		NOT checkBottom OR_ELSE InsertionQuality(
			suctions:= suctionBottom, 
			insertionMaterial:= loadedMaterials[Surface.BOTTOM], 
			recipeMaterial:= materialsArr[iPair].bottom)
	);
*)
END_METHOD

END_FUNCTION_BLOCK

// ---- DUTs/Hardware/Big Machines/StrapMachine.TcPOU
FUNCTION_BLOCK StrapMachine
VAR_INPUT
	bEnable : BOOL;
	extSafety : BOOL;
END_VAR
VAR_OUTPUT
	enable AT %Q* : BOOL;
	execute AT %Q* : BOOL;
	reset AT %Q* : BOOL;
	
	error AT %I* : BOOL;
	ready AT %I* : BOOL;
	//busy (*AT %I**) : BOOL;
	done AT %I* : BOOL;
	home AT %I* : BOOL;
	
	timeout : BOOL;
	
	atBundleLevel AT %I* : BOOL;
END_VAR
VAR	
	holdPost : TON;
	timeoutDelay : TON;
	resetDelay : TP;
	
	start : BOOL;
	step : (SETUP, RUN, WAIT);
END_VAR
VAR_STAT CONSTANT
	maxDelay : TIME := T#30S;
	pulseWidth : TIME := T#500MS;
END_VAR

holdPost(IN:= , PT:= pulseWidth, Q=> , ET=> );
timeoutDelay(IN:= (step > 0), PT:= maxDelay, Q=> timeout, ET=> );

resetDelay(IN:= error AND NOT resetDelay.Q , PT:= pulseWidth, Q=> , ET=> );
reset := resetDelay.Q AND (resetDelay.ET > resetDelay.PT/2);

IF timeoutDelay.Q THEN
	timeoutDelay.IN := FALSE;
	timeout := TRUE;
	//busy := FALSE;
	
	start := FALSE;
	step := SETUP;
END_IF

//enable := bEnable AND robot1.strapSafetyIn AND robot2.strapSafetyIn;
//enable := bEnable AND robot1StrapSafety AND robot2StrapSafety;
enable := bEnable AND extSafety;

CASE step OF
	SETUP:
		IF error THEN
			enable := FALSE;
			execute := FALSE;
			RETURN;
		END_IF
		
		IF start AND enable (*AND ready*) THEN //strapping does not start if error
			start := FALSE;
			step := RUN;
		END_IF
	
	RUN:
		IF NOT execute THEN
			execute := TRUE;
			RETURN; //keeps execute TRUE for at least 1 cycle
		END_IF
		
		IF execute AND NOT ready (*AND NOT home*) THEN
			execute := FALSE;
			step := WAIT;
		END_IF
		
	WAIT: //due to the use of DC motors instead of stepper motors in the machine, a short delay is required before next strap
		IF home THEN
			holdPost.IN := TRUE;
			execute := FALSE;
			enable := FALSE;
		END_IF
		
		IF holdPost.Q THEN
			holdPost.IN := FALSE;
			step := 0;
		END_IF
		
END_CASE

(*
executePulse(IN:= , PT:= pulseTime, Q=> , ET=> );
execute := executePulse.IN AND NOT executePulse.Q;

IF executePulse.Q THEN
	executePulse.IN := FALSE;
END_IF


resetPulse(IN:= , PT:= pulseTime, Q=> , ET=> );
StrapMachineST.reset := resetPulse.IN AND NOT resetPulse.Q;

IF resetPulse.Q THEN
	executePulse.IN := FALSE;
END_IF

ready := enable AND NOT execute AND NOT StrapMachineST.reset AND NOT error AND home;
*)

METHOD clear : BOOL
VAR_INPUT
END_VAR
(*
reset should be continuously called until machine returns evidence that it is ready again
machine is expected to not respond to reset signals if it is already in an idle state
*)
END_METHOD

METHOD strap : BOOL
VAR_INPUT
END_VAR
//IF ready AND NOT busy AND NOT error THEN
	//busy := TRUE;
	//start := TRUE;
	//strap := TRUE;
//END_IF

start := TRUE;
END_METHOD

END_FUNCTION_BLOCK

// ---- Sections/A21b - Wood Bunk/AOIs/AOI_StageWoodBunk.TcPOU
FUNCTION_BLOCK AOI_StageWoodBunk
VAR_INPUT
	execute : BOOL;
END_VAR
VAR_IN_OUT CONSTANT
	sectionID : SectionEnum;
END_VAR
VAR_IN_OUT
	robot : RobotA21;
	table : StagingTable;
	magazine : SkidMagazine;
END_VAR
VAR_INPUT
	slot : INT;
	material : STRING;
END_VAR
VAR_OUTPUT
	busy : BOOL;
	done : BOOL; //this done signal stays on until next execution
	error : BOOL;
	
	recovery : BOOL;
	failCounter : INT;
	
	donePulse : BOOL; //this done signal only stays on for 1 cycle after completion
END_VAR
VAR
	run : BOOL;
	trigger : R_TRIG;	
	doneTrigger : R_TRIG;
	
	column : INT;
	step : (IDLE, PREP_ROBOT, GET_FROM_MAGAZINE, PLACE_ON_TABLE, COMPLETE);
END_VAR
VAR CONSTANT
	suctionDistance : INT := 10;
END_VAR

{warning disable C0371}
{warning disable C0195}
(*
IF error THEN
	step := IDLE;
END_IF
*)
trigger(CLK:= execute, Q=> );
doneTrigger(CLK:= done, Q=> donePulse);

busy := trigger.Q OR step > 0;

IF step > IDLE AND_THEN NOT preExecution() THEN //conditions to track before execution
	RETURN;
END_IF

//follow the template as is
CASE step OF
	IDLE:
		IF trigger.Q THEN //reset outputs
			done := FALSE;
			error := FALSE;
			recovery := FALSE;
			
			step := PREP_ROBOT;
		END_IF
		
	PREP_ROBOT:
		robot.clearCommand();
		IF robot.Ready THEN
			step := GET_FROM_MAGAZINE;
		END_IF
	
	GET_FROM_MAGAZINE: //grab from magazine
		IF NOT magazine.findSlot(material := material, index => column) THEN
			error := TRUE;
			RETURN;
		END_IF
		
		IF robot.eoatDistance < suctionDistance THEN //robot is grabbing material
			robot.HoldMaterial := magazine.getSlot(i := column);
		END_IF
		
		IF robot.Done THEN
			step := COMPLETE;
			RETURN;
		END_IF
		
		robot.setGroup(group := 1, value := TaskA21.STAGE_BUNK);
		robot.setGroup(group := 2, value := column);
		robot.setGroup(group := 3, value := slot);

	COMPLETE: //check here if staging is successful or needs to be repeated
		robot.clearCommand();
		
		IF table.isOccupied(slot) THEN
			table.place(i := slot, materialID := robot.HoldMaterial);
			robot.HoldMaterial := '';
			
			failCounter := 0;
			done := TRUE;
		ELSE
			failCounter := failCounter + 1;
		END_IF
		
		step := 0;
		
END_CASE

METHOD PRIVATE preExecution : BOOL
VAR_INPUT
END_VAR
{warning disable C0371}

IF slot < 1 THEN //out of bounds for staging table
	error := TRUE;
	RETURN;
ELSIF table.isFull() OR slot > 10 OR material = '' OR table.getSlot(i := slot, error => ) = material THEN
	done := TRUE;
	RETURN;
END_IF

IF //robot must be ready before execution
	robot.error OR 
	robot.reservation <> sectionID OR 
	robot.tool <> sectionID
THEN
	error := TRUE;
	RETURN;
END_IF

preExecution := TRUE;
END_METHOD

METHOD reset : BOOL
VAR_INPUT
END_VAR
VAR
	temp : AOI_StageWoodBunk;
END_VAR
//(*
done := FALSE;
error := FALSE;
recovery := FALSE;
slot := 0;
step := 0;

failCounter := 0;
//*)
//THIS^ := temp;
END_METHOD

END_FUNCTION_BLOCK

// ---- POUs/Helper Functions/Hardware Modules/SuctionQuality.TcPOU
FUNCTION SuctionQuality : BOOL
VAR_IN_OUT
	suctions : ARRAY[*] OF SuctionPad;
END_VAR
VAR
	i : DINT;
	
	failedPads : INT;
	numPads : INT;
END_VAR

FOR i:=LOWER_BOUND(suctions, 1) TO UPPER_BOUND(suctions, 1) BY 1 DO
	IF suctions[i].enable THEN
		numPads := numPads + 1;
		IF NOT suctions[i].occupied THEN
			failedPads := failedPads + 1;
		END_IF
	END_IF
	
END_FOR

SuctionQuality := TRUE;
	//failedPads <= numPads/2;

END_FUNCTION

// ---- COMs/Local Devices/EcNetwork.TcPOU
FUNCTION_BLOCK EcNetwork
VAR_INPUT
	enable : BOOL;
	netID : T_AmsNetId; //AmsNetID of the EtherCAT master node (NIC, EK1200, etc)
END_VAR
VAR_OUTPUT 
	slaves : ARRAY[0..EC_MAX_SLAVES] OF ST_EcSlaveConfigData; //devices
	slaveStates : ARRAY[0..EC_MAX_SLAVES] OF ST_EcSlaveState; //device states
	
	//start-end indexes for each subarea to access
	deviceIndexesA21 : ARRAY[0..1] OF DINT;
	deviceIndexesA22 : ARRAY[0..1] OF DINT;
	deviceIndexesA23 : ARRAY[0..1] OF DINT;
	deviceIndexesA24 : ARRAY[0..1] OF DINT;
	deviceIndexesA25 : ARRAY[0..1] OF DINT;
	deviceIndexesA26 : ARRAY[0..1] OF DINT;
END_VAR
VAR_OUTPUT
	numSlaves : DINT; //nSlaves must be cast from UINT to DINT in order to end iteration at -1 if there are no slaves
	
	diagnosticsError : BOOL;
	errorInit : BOOL;
	errorPreop : BOOL;
	errorBootstrap : BOOL;
	errorSafeop : BOOL;
	
	operational : BOOL;
END_VAR
VAR
	fbEcGetAllSlaveStates : FB_EcGetAllSlaveStates;
	fbEcGetConfiguredSlaves : FB_EcGetConfSlaves;
	
	i : DINT;
END_VAR

blocks();

diagnosticsError := fbEcGetAllSlaveStates.bError OR fbEcGetConfiguredSlaves.bError;
errorInit := FALSE;
errorPreop := FALSE;
errorBootstrap := FALSE;
errorSafeop := FALSE;

CheckEcNetwork(
	ecDeviceStates:= slaveStates, 
	ecIndex0:= 0, 
	ecIndex1:= numSlaves-1, 
	errorInit=> errorInit, 
	errorPreop=> errorPreop, 
	errorBootstrap=> errorBootstrap, 
	errorSafeop=> errorSafeop, 
	error=> , 
	operational=> operational);

distributeIndexes(slavePrefix:= 'A21', firstIndex=> deviceIndexesA21[0], lastIndex=> deviceIndexesA21[1]);
distributeIndexes(slavePrefix:= 'A22', firstIndex=> deviceIndexesA22[0], lastIndex=> deviceIndexesA22[1]);
distributeIndexes(slavePrefix:= 'A23', firstIndex=> deviceIndexesA23[0], lastIndex=> deviceIndexesA23[1]);
distributeIndexes(slavePrefix:= 'A24', firstIndex=> deviceIndexesA24[0], lastIndex=> deviceIndexesA24[1]);
distributeIndexes(slavePrefix:= 'A25', firstIndex=> deviceIndexesA25[0], lastIndex=> deviceIndexesA25[1]);
distributeIndexes(slavePrefix:= 'A26', firstIndex=> deviceIndexesA26[0], lastIndex=> deviceIndexesA26[1]);

METHOD PRIVATE blocks : BOOL
VAR_INST // added by the converter: edge detectors and wires of the graphical bodies
    _w1, _w2 : BOOL;
END_VAR
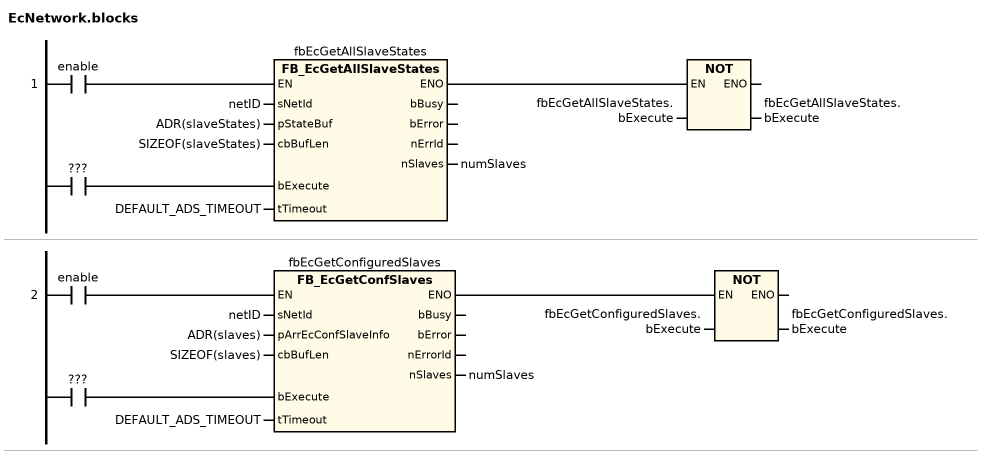
// NETWORK 1
_w1 := enable;
IF _w1 THEN
    fbEcGetAllSlaveStates(
        sNetId := netID,
        pStateBuf := ADR(slaveStates),
        cbBufLen := SIZEOF(slaveStates),
        tTimeout := DEFAULT_ADS_TIMEOUT,
        nSlaves => numSlaves); // FB_EcGetAllSlaveStates
END_IF
IF _w1 THEN fbEcGetAllSlaveStates.bExecute := NOT fbEcGetAllSlaveStates.bExecute; END_IF

// NETWORK 2
_w2 := enable;
IF _w2 THEN
    fbEcGetConfiguredSlaves(
        sNetId := netID,
        pArrEcConfSlaveInfo := ADR(slaves),
        cbBufLen := SIZEOF(slaves),
        tTimeout := DEFAULT_ADS_TIMEOUT,
        nSlaves => numSlaves); // FB_EcGetConfSlaves
END_IF
IF _w2 THEN fbEcGetConfiguredSlaves.bExecute := NOT fbEcGetConfiguredSlaves.bExecute; END_IF
END_METHOD

METHOD PRIVATE distributeIndexes : BOOL
VAR_INPUT
	slavePrefix : STRING;
END_VAR
VAR_OUTPUT
	firstIndex : DINT;
	lastIndex : DINT := -1; //no iteration if last index < first index
END_VAR
VAR
	firstIndexSet : BOOL;
	i : DINT;
END_VAR
FOR i:=0 TO numSlaves-1 BY 1 DO	
	IF NOT firstIndexSet THEN
		firstIndexSet := TRUE;
		firstIndex := i;
		
	ELSIF FIND(slaves[i].sName, slavePrefix) = 0 THEN
		RETURN;
		
	END_IF
	
	lastIndex := i;
	
END_FOR
END_METHOD

END_FUNCTION_BLOCK

// ---- POUs/Helper Functions/Hardware Modules/CheckEcNetwork.TcPOU
FUNCTION CheckEcNetwork : BOOL
VAR_IN_OUT
	ecDeviceStates : ARRAY[*] OF ST_EcSlaveState;
END_VAR
VAR_INPUT
	ecIndex0, ecIndex1 : DINT;
END_VAR
VAR_OUTPUT
	errorInit : BOOL;
	errorPreop : BOOL;
	errorBootstrap : BOOL;
	errorSafeop : BOOL;
	
	error : BOOL;
	operational : BOOL;
END_VAR
VAR
	i : DINT;
END_VAR

CheckEcNetwork := 
	InRange(v1:= 0, v2:= EC_MAX_SLAVES, value:= ecIndex0, inclusive:= TRUE) AND
	InRange(v1:= 0, v2:= EC_MAX_SLAVES, value:= ecIndex1, inclusive:= TRUE) AND
	ecIndex0 < ecIndex1;

FOR i:=ecIndex0 TO ecIndex1 BY 1 DO
	
	CASE ecDeviceStates[i].deviceState OF
		EC_DEVICE_STATE_INIT:			errorInit := TRUE;
		EC_DEVICE_STATE_PREOP:			errorPreop := TRUE;
		EC_DEVICE_STATE_BOOTSTRAP:		errorBootstrap := TRUE;
		EC_DEVICE_STATE_SAFEOP:			errorSafeop := TRUE;
	END_CASE
	
END_FOR

error := 
	errorInit OR 
	errorPreop OR
	errorBootstrap OR
	errorSafeop OR
	NOT CheckEcNetwork;
	
operational := NOT error;

END_FUNCTION

// ---- POUs/Helper Functions/General/InRange.TcPOU
FUNCTION InRange : BOOL
VAR_INPUT
	v1 : LREAL;
	v2 : LREAL;
	value : LREAL;
	
	inclusive : BOOL;
END_VAR
VAR
	lower : LREAL;
	upper : LREAL;
END_VAR

lower := MIN(v1, v2);
upper := MAX(v1, v2);

IF inclusive THEN
	InRange := (value >= lower AND value <= upper);
ELSE
	InRange := (value > lower AND value < upper);
END_IF

END_FUNCTION

// ---- HARDWARE_DISTRUBUTION/A21.TcPOU
FUNCTION_BLOCK A21 EXTENDS GenericSubarea
VAR_IN_OUT
	sectionCIP : ChipboardEx;
	sectionWB : WoodBunkEx;
END_VAR
VAR //conveyor arrays
	conveyorsCIP : ARRAY[1..3] OF POINTER TO ConveyorSC;
	conveyorsWB : ARRAY[1..1] OF POINTER TO ConveyorSC;
END_VAR
VAR //hardware
	robot1, robot2 : RobotA21;
	
	toolStorageA21Left, toolStorageA21Right : A21ToolStorage;
	
	skidA21Left, skidA21Right : SkidMagazine;
	magazineA21Left, magazineA21Right : SkidMagazine;
	stagingTableLeft, stagingTableRight : StagingTable;
	strapperA21 : StrapMachine;
	
	centeringSliderA21 : ServoNC;
	
	horizontalDriveA21Left, horizontalDriveA21Right : AirPiston := (
		limitSensorDefaultState := FALSE,
		useBrake := FALSE);
	
	verticalDriveA21Left, verticalDriveA21Right : ClearLinkMC := (
		limitSensorDefaultState := TRUE, 
		homingDirectionOut := TRUE, //outwards (up)
		minPosition := 0,
		displacementPerRotation := 1,
		unitsPerPulse := 8000); //0.1x gearbox, 10 revs/pulse to compensate
		
	insertionA21Left, insertionA21Right : Insertion;
	
	pistonA21Bottom : SimplePiston;
	
	suctionA21Top : ARRAY[1..3] OF SuctionPad;
	suctionA21Left : ARRAY[1..4] OF SuctionPad;
	suctionA21Right : ARRAY[1..4] OF SuctionPad; 
	suctionA21Bottom : ARRAY[1..2] OF SuctionPad;
END_VAR
VAR //different material holders have different capacities, so arrays of slots are declared externally and passed in
	skidSlotsA21Left, skidSlotsA21Right AT %M* : ARRAY[1..2] OF MaterialSlot; //%M* declaration overrides %I* and %Q* attributes
	magazineSlotsA21Left, magazineSlotsA21Right AT %M* : ARRAY[1..15] OF MaterialSlot;
	tableSlotsA21Left, tableSlotsA21Right : ARRAY[1..10] OF MaterialSlot;
END_VAR
VAR //statuses and alarms
	stackLightCIP : PMLStackLight; //chipboard stack light
	stackLightWB : PMLStackLight; //wood bunk stack light
	
	panelPowerOn : BOOL;
	safetyOk : BOOL;
	airPressureOk : BOOL;
END_VAR

SUPER^();

METHOD PROTECTED callHardware : BOOL
{warning disable C0371}

robot1(strapSafety := (NOT strapperA21.enable AND NOT strapperA21.execute AND strapperA21.home));	
robot2(strapSafety := (NOT strapperA21.enable AND NOT strapperA21.execute AND strapperA21.home));

skidA21Left(slots := skidSlotsA21Left);
skidA21Right(slots := skidSlotsA21Right);

stagingTableLeft(slots := tableSlotsA21Left);
stagingTableRight(slots := tableSlotsA21Right);

magazineA21Left(slots := magazineSlotsA21Left);
magazineA21Right(slots := magazineSlotsA21Right);

strapperA21(extSafety := robot1.strapSafetyIn AND robot2.strapSafetyIn);

verticalDriveA21Left(bEnable := TRUE);
verticalDriveA21Right(bEnable := TRUE);
horizontalDriveA21Left(bEnable := TRUE);
horizontalDriveA21Right(bEnable := TRUE);

insertionA21Left(
	slider:= verticalDriveA21Left, 
	screw:= horizontalDriveA21Left, 
	contact=> , 
	active=> , 
	error=> , 
	home=> , 
	homingComplete=> , 
	sliderPos=> );
	
insertionA21Right(
	slider:= verticalDriveA21Right, 
	screw:= horizontalDriveA21Right, 
	contact=> , 
	active=> , 
	error=> , 
	home=> , 
	homingComplete=> , 
	sliderPos=> );

pistonA21Bottom();

stackLightCIP(
	pmlState:= sectionCIP.pmlState, 
	lowMaterial:= , 
	materialExhausted:= , 
	red=> , 
	yellow=> , 
	blue=> , 
	green=> );
	
stackLightWB(
	pmlState:= sectionWB.pmlState, 
	lowMaterial:= , 
	materialExhausted:= , 
	red=> , 
	yellow=> , 
	blue=> , 
	green=> );

(*
tempLeft := TO_INT(BoolPtrArrayToInteger(arr := stagingTableLeft.occupied, lowerBound := 1, upperBound := 10));
tempLeft.15 := NOT strapperA21.bEnable AND NOT strapperA21.execute;
robot1.setGroup(group := 8, value := tempLeft);

tempRight := TO_INT(BoolPtrArrayToInteger(arr := stagingTableRight.occupied, lowerBound := 1, upperBound := 10));
tempRight.15 := NOT strapperA21.bEnable AND NOT strapperA21.execute;
robot2.setGroup(group := 8, value := tempRight);

*)
END_METHOD

METHOD PROTECTED runModules : BOOL
VAR_INPUT
END_VAR
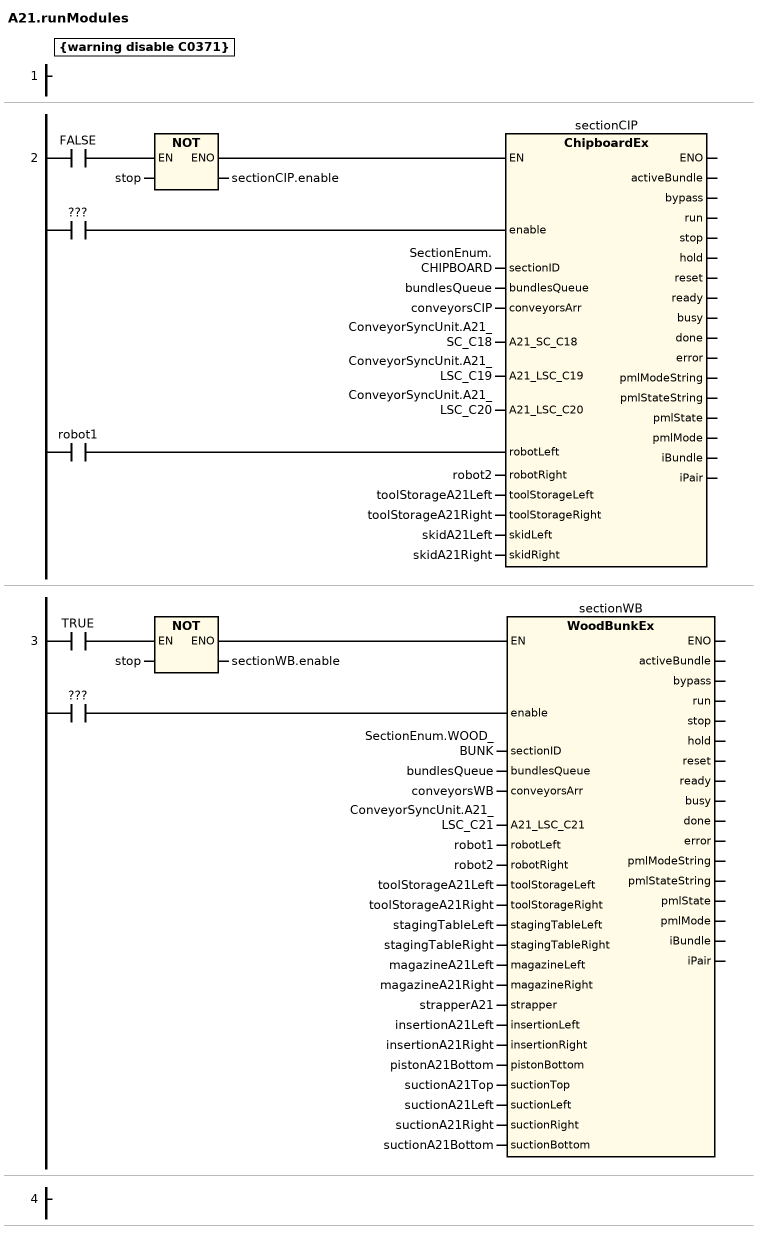
// NETWORK 1
// label: {warning disable C0371}

// NETWORK 2
IF FALSE THEN sectionCIP.enable := NOT stop; END_IF
IF FALSE THEN
    sectionCIP(
        sectionID := SectionEnum.CHIPBOARD,
        bundlesQueue := bundlesQueue,
        conveyorsArr := conveyorsCIP,
        A21_SC_C18 := ConveyorSyncUnit.A21_SC_C18,
        A21_LSC_C19 := ConveyorSyncUnit.A21_LSC_C19,
        A21_LSC_C20 := ConveyorSyncUnit.A21_LSC_C20,
        robotLeft := robot1,
        robotRight := robot2,
        toolStorageLeft := toolStorageA21Left,
        toolStorageRight := toolStorageA21Right,
        skidLeft := skidA21Left,
        skidRight := skidA21Right); // ChipboardEx
END_IF

// NETWORK 3
sectionWB.enable := NOT stop;
sectionWB(
    sectionID := SectionEnum.WOOD_BUNK,
    bundlesQueue := bundlesQueue,
    conveyorsArr := conveyorsWB,
    A21_LSC_C21 := ConveyorSyncUnit.A21_LSC_C21,
    robotLeft := robot1,
    robotRight := robot2,
    toolStorageLeft := toolStorageA21Left,
    toolStorageRight := toolStorageA21Right,
    stagingTableLeft := stagingTableLeft,
    stagingTableRight := stagingTableRight,
    magazineLeft := magazineA21Left,
    magazineRight := magazineA21Right,
    strapper := strapperA21,
    insertionLeft := insertionA21Left,
    insertionRight := insertionA21Right,
    pistonBottom := pistonA21Bottom,
    suctionTop := suctionA21Top,
    suctionLeft := suctionA21Left,
    suctionRight := suctionA21Right,
    suctionBottom := suctionA21Bottom); // WoodBunkEx

// NETWORK 4
END_METHOD

METHOD PROTECTED setupHardware : BOOL
VAR
	iWoodBunkSlot : WoodBunk;
	iChipboardSlot : Chipboard;
	i : INT;
END_VAR
FOR iWoodBunkSlot:=1 TO WoodBunk.size-1 BY 1 DO //init wood bunk magazine slots
	magazineA21Left.setSlot(i := iWoodBunkSlot, material := TO_STRING(iWoodBunkSlot), error => );
	magazineA21Right.setSlot(i := iWoodBunkSlot, material := TO_STRING(iWoodBunkSlot), error => );
END_FOR

//--------------------------------------------------

FOR iChipboardSlot:=1 TO Chipboard.size-1 BY 1 DO //init chipboard skid slots
	skidA21Left.setSlot(i := iChipboardSlot, material := TO_STRING(iChipboardSlot), error => );
	skidA21Right.setSlot(i := iChipboardSlot, material := TO_STRING(iChipboardSlot), error => );
END_FOR

//--------------------------------------------------

FOR i:=1 TO CONSTS.maxQueue BY 1 DO //get wood bunk magazine + chipboard skid availability from robot1 and robot2
	{warning disable C0195}
	skidA21Left.setOccupancy( i := i, occupancy := IntegerBitAccess(robot1.inputs[4], i-1) );
	skidA21Right.setOccupancy( i := i, occupancy := IntegerBitAccess(robot2.inputs[4], i-1) );

	magazineA21Left.setOccupancy( i := i, occupancy := IntegerBitAccess(robot1.inputs[3], i-1) );
	magazineA21Right.setOccupancy( i := i, occupancy := IntegerBitAccess(robot2.inputs[3], i-1) );
END_FOR

//--------------------------------------------------
conveyorsCIP[1] := ADR(ConveyorSyncUnit.A21_SC_C18);
conveyorsCIP[2] := ADR(ConveyorSyncUnit.A21_LSC_C19);
conveyorsCIP[3] := ADR(ConveyorSyncUnit.A21_LSC_C20);

conveyorsWB[1] := ADR(ConveyorSyncUnit.A21_LSC_C21);
END_METHOD

END_FUNCTION_BLOCK

// ---- HARDWARE_DISTRUBUTION/GenericSubarea.TcPOU
FUNCTION_BLOCK ABSTRACT GenericSubarea
VAR_IN_OUT
	bundlesQueue : ARRAY[*] OF Bundle;
	
	//ecDevices : ARRAY[0..EC_MAX_SLAVES] OF ST_EcSlaveConfigData; //devices
	ecDeviceStates : ARRAY[*] OF ST_EcSlaveState; //device states
END_VAR
VAR_INPUT
	ecIndex0, ecIndex1 : DINT;
END_VAR
VAR_OUTPUT //controls
	stop AT %I* : BOOL;
	
	ready : BOOL;
	active : BOOL;
	error : BOOL;
	
	ecNetworkError : BOOL;
END_VAR

CheckEcNetwork(
	ecDeviceStates:= ecDeviceStates, 
	ecIndex0:= ecIndex0, 
	ecIndex1:= ecIndex1, 
	errorInit=> , 
	errorPreop=> , 
	errorBootstrap=> , 
	errorSafeop=> , 
	error=> ecNetworkError, 
	operational=> );
	
callHardware();

setupHardware();

runModules();

callHardware();

METHOD PROTECTED ABSTRACT callHardware : BOOL
VAR_INPUT
END_VAR
END_METHOD

METHOD PROTECTED ABSTRACT runModules : BOOL
VAR_INPUT
END_VAR
END_METHOD

METHOD PROTECTED ABSTRACT setupHardware : BOOL
VAR_INPUT
END_VAR
END_METHOD

END_FUNCTION_BLOCK

// ---- DUTs/Hardware/Insertion Package/Drives/AirPiston.TcPOU
FUNCTION_BLOCK AirPiston EXTENDS FBA_Drive IMPLEMENTS I_ContinuousDrive
VAR_OUTPUT
	valveExtend AT %Q* : BOOL;
	valveRetract AT %Q* : BOOL;
END_VAR
VAR //constructor
	useBrake : BOOL; //optional - set to FALSE if retraction brake pulse is not required
END_VAR
VAR
	mode : (HOLD, IN, OUT, BRAKE);
	brakePulse : TP; //generates the retraction pulse
END_VAR
VAR_STAT CONSTANT
	brakeWidth : TIME := T#650MS;
END_VAR

IF NOT bEnable THEN
	stop();
	RETURN;
END_IF

brakePulse(IN:= , PT:= brakeWidth, Q=> , ET=> ); //reversal to act as brake
brakePulse.IN := brakePulse.IN AND brakePulse.Q; //automatically turn off pulse

override(); //alters the mode to prevent exceeding limits

CASE mode OF
	HOLD:
		valveExtend := FALSE;
		valveRetract := FALSE;
		
	IN:
		valveExtend := TRUE;
		valveRetract := FALSE;
		
	OUT:
		valveExtend := FALSE;
		valveRetract := TRUE;
		
	BRAKE: //coasts past inner limit, then slides back
		valveExtend := FALSE;
		valveRetract := TRUE;
		
		IF AtHome THEN
			mode := HOLD;
		END_IF
		
END_CASE

valveRetract := valveRetract OR brakePulse.Q; //from mode or brake

PROPERTY Active : BOOL
GET
Active :=
	mode <> HOLD AND
	valveExtend OR valveRetract;
END_GET
END_PROPERTY

PROPERTY Error : BOOL
GET
END_GET
END_PROPERTY

METHOD extend : BOOL
VAR_INPUT
END_VAR
IF mode <> BRAKE THEN
	mode := IN;
END_IF
END_METHOD

METHOD homingSequence : BOOL
CASE step OF
	Homing.IDLE:
		step := Homing.START;
		
	Homing.START:
		IF AtHome THEN //if reached home
			step := Homing.DONE;
		ELSE
			mode := OUT;
		END_IF
		
	Homing.DONE:
		mode := HOLD;
		homingComplete := TRUE;
		homingSequence := TRUE;		
	
END_CASE
END_METHOD

{attribute 'TcRpcEnable'}
METHOD moveContinuous : BOOL
VAR_INPUT
	direction : MC_Direction;
END_VAR
IF direction = MC_Positive_Direction THEN
	retract();
ELSIF direction = MC_Negative_Direction THEN
	extend();
END_IF
END_METHOD

METHOD PRIVATE override : BOOL
VAR_INPUT
END_VAR
IF brakePulse.Q THEN
	mode := HOLD;
END_IF

IF AtHome AND (valveRetract OR mode = OUT) THEN
	mode := HOLD;
	
ELSIF AtInnerLimit AND (valveExtend OR mode = IN) THEN	
	brakePulse.IN := useBrake;
	mode := HOLD;
END_IF


IF NOT bEnable THEN
	stop();
END_IF
END_METHOD

METHOD reset : BOOL
VAR_INPUT
END_VAR
stop();
END_METHOD

METHOD retract : BOOL
VAR_INPUT
END_VAR
IF mode <> BRAKE THEN
	mode := OUT;
END_IF
END_METHOD

METHOD stop : BOOL
VAR_INPUT
END_VAR
valveExtend := FALSE;
valveRetract := FALSE;
mode := HOLD;
END_METHOD

METHOD toHome : BOOL
VAR_INPUT
END_VAR
mode := OUT;
END_METHOD

END_FUNCTION_BLOCK

// ---- DUTs/Hardware/PMLStackLight.TcPOU
FUNCTION_BLOCK PMLStackLight
VAR_INPUT
	pmlState : E_PMLState;
	lowMaterial : BOOL;
	materialExhausted : BOOL;
END_VAR
VAR_OUTPUT
	red AT %M* : BOOL;
	yellow AT %M* : BOOL;
	blue AT %M* : BOOL;
	green AT %M* : BOOL;
END_VAR
VAR_STAT //flashing is sychronized between all instances
	redPulse : TP;
	yellowPulse : TP;
	bluePulse : TP;
	greenPulse : TP;
	
	flashingRed : BOOL;
	flashingYellow : BOOL;
	flashingBlue : BOOL;
	flashingGreen : BOOL;
END_VAR
VAR_STAT CONSTANT
	flashWidth : TIME := T#1500MS;
END_VAR

redPulse(IN:= NOT redPulse.Q, PT:= flashWidth, Q=> , ET=> );
yellowPulse(IN:= NOT yellowPulse.Q, PT:= flashWidth, Q=> , ET=> );
bluePulse(IN:= NOT bluePulse.Q, PT:= flashWidth, Q=> , ET=> ); //material status light
greenPulse(IN:= NOT greenPulse.Q, PT:= flashWidth, Q=> , ET=> );

flashingRed := redPulse.Q AND redPulse.ET < flashWidth/2;
flashingYellow := yellowPulse.Q AND yellowPulse.ET < flashWidth/2;
flashingBlue := bluePulse.Q AND bluePulse.ET < flashWidth/2;
flashingGreen := greenPulse.Q AND greenPulse.ET < flashWidth/2;

blue := materialExhausted OR (lowMaterial AND flashingBlue);

//stack light sequences
CASE pmlState OF
	0: //nothing
	ePMLState_Stopping:			ps_Stopping();
	ePMLState_Stopped:			ps_Stopped();
    ePMLState_Resetting:		ps_Resetting();
	ePMLState_Idle:				ps_Idle();
	ePMLState_Starting:			ps_Starting();
	ePMLState_Execute:			ps_Execute();
	ePMLState_Completing:		ps_Completing();
	ePMLState_Complete:			ps_Complete();
	ePMLState_Holding:			ps_Holding();
	ePMLState_Held:				ps_Held();
	ePMLState_Unholding:		ps_Unholding();
	ePMLState_Suspended:		ps_Suspended();
	ePMLState_Suspending:		ps_Suspending();
	ePMLState_Unsuspending:		ps_Unsuspending();
	ePMLState_Aborting:			ps_Aborting();
	ePMLState_Aborted:			ps_Aborted();
	ePMLState_Clearing:			ps_Clearing();
END_CASE

METHOD PROTECTED ps_Aborted : BOOL
VAR_INPUT
END_VAR
red := flashingRed;
yellow := FALSE;
green := FALSE;
END_METHOD

METHOD PROTECTED ps_Aborting : BOOL
VAR_INPUT
END_VAR
red := flashingRed;
yellow := FALSE;
green := FALSE;
END_METHOD

METHOD PROTECTED ps_Clearing : BOOL
VAR_INPUT
END_VAR
red := flashingRed;
yellow := FALSE;
green := FALSE;
END_METHOD

METHOD PROTECTED ps_Complete : BOOL
VAR_INPUT
END_VAR
red := TRUE;
yellow := FALSE;
green := FALSE;
END_METHOD

METHOD PROTECTED ps_Completing : BOOL
VAR_INPUT
END_VAR
red := FALSE;
yellow := FALSE;
green := TRUE;
END_METHOD

METHOD PROTECTED ps_Execute : BOOL
VAR_INPUT
END_VAR
VAR_OUTPUT
	error : BOOL;
END_VAR
red := FALSE;
yellow := FALSE;
green := TRUE;
END_METHOD

METHOD PROTECTED ps_Held : BOOL
VAR_INPUT
END_VAR
red := FALSE;
yellow := FALSE;
green := FALSE;
END_METHOD

METHOD PROTECTED ps_Holding : BOOL
VAR_INPUT
END_VAR
red := FALSE;
yellow := FALSE;
green := FALSE;
END_METHOD

METHOD PROTECTED ps_Idle : BOOL
VAR_INPUT
END_VAR
red := FALSE;
yellow := FALSE;
green := flashingGreen;
END_METHOD

METHOD PROTECTED ps_Resetting : BOOL
VAR_INPUT
END_VAR
red := TRUE;
yellow := FALSE;
green := FALSE;
END_METHOD

METHOD PROTECTED ps_Starting : BOOL
VAR_INPUT
END_VAR
red := FALSE;
yellow := FALSE;
green := TRUE;
END_METHOD

METHOD PROTECTED ps_Stopped : BOOL
VAR_INPUT
END_VAR
red := TRUE;
yellow := FALSE;
green := FALSE;
END_METHOD

METHOD PROTECTED ps_Stopping : BOOL
VAR_INPUT
END_VAR
red := TRUE;
yellow := FALSE;
green := FALSE;
END_METHOD

METHOD PROTECTED ps_Suspended : BOOL
VAR_INPUT
END_VAR
red := FALSE;
yellow := TRUE;
green := TRUE;
END_METHOD

METHOD PROTECTED ps_Suspending : BOOL
VAR_INPUT
END_VAR
red := FALSE;
yellow := TRUE;
green := TRUE;
END_METHOD

METHOD PROTECTED ps_Unholding : BOOL
VAR_INPUT
END_VAR
red := FALSE;
yellow := FALSE;
green := FALSE;
END_METHOD

METHOD PROTECTED ps_Unsuspending : BOOL
VAR_INPUT
END_VAR
red := FALSE;
yellow := TRUE;
green := FALSE;
END_METHOD

METHOD PROTECTED setStackLights : BOOL
VAR_INPUT
	redLight : BOOL;
	yellowLight : BOOL;
	blueLight : BOOL;
	greenLight : BOOL;
END_VAR
red := redLight;
yellow := yellowLight;
blue := blueLight;
green := greenLight;
END_METHOD

END_FUNCTION_BLOCK

// ---- HARDWARE_DISTRUBUTION/ConveyorSyncUnit.TcPOU
PROGRAM ConveyorSyncUnit
VAR_OUTPUT
	A24_LRC_C02 	: Conveyor; //these conveyoors move bundles from A2.7 to A2.4
	A24_LRC_C04 	: Conveyor;
	A24_LRC_C06	 	: Conveyor;
	A24_LRC_C08 	: Conveyor;
	A24_LRC_C10 	: Conveyor;
	A24_LRC_C12 	: Conveyor;
	
	A24_SC_C01 		: ConveyorSC; //these conveyors move bundles on A2.4 forward down the cell
	A24_SC_C03 		: ConveyorSC;
	A24_SC_C05 		: ConveyorSC;
	A24_SC_C07 		: ConveyorSC;
	A24_SC_C09 		: ConveyorSC;
	A24_SC_C11 		: ConveyorSC;
	A24_SC_C13 		: ConveyorSC;
	
	A23_LSC_C14 	: ConveyorLSC;
	
	A22_SC_C15 		: ConveyorSC;
	A22_LSC_C16 	: ConveyorLSC;
	A22_LSC_C17 	: ConveyorLSC;
	
	A21_SC_C18 		: ConveyorSC;
	A21_LSC_C19 	: ConveyorLSC;
	A21_LSC_C20 	: ConveyorLSC;
	A21_LSC_C21 	: ConveyorLSC;
	
	A25_SC_C22 		: ConveyorSC;
	A25_SC_C24 		: ConveyorSC;
	A25_SC_C26 		: ConveyorSC;
	A25_SC_C28 		: ConveyorSC;
	A25_SC_C30 		: ConveyorSC;
	
	A25_LSC_C23 	: ConveyorLSC; //these conveyors move the bundle sideways onto the output buffers
	A25_LSLCC_C25 	: ConveyorLSC;
	A25_LSLCC_C27 	: ConveyorLSC;
	A25_LSC_C29 	: ConveyorLSC;
	A25_SC_C31 		: ConveyorSC;
	A25_SC_C32 		: ConveyorSC;
	A25_SC_C33 		: ConveyorSC;
	A25_SC_C34 		: ConveyorSC;
	A25_SC_C35 		: ConveyorSC;
	A25_SC_C36 		: ConveyorSC;
	A25_SC_C37 		: ConveyorSC;
	A25_SC_C38 		: ConveyorSC;
END_VAR
VAR
	cellConveyors : ARRAY[1..numCellConveyors] OF POINTER TO ConveyorSC;
	receiverConveyors : ARRAY[1..numReceiverConveyors] OF POINTER TO ConveyorSC;
	outputConveyors : ARRAY[1..numOutputConveyors] OF POINTER TO ConveyorSC;
	
	spoolTimer : TON;
	i : DINT := 1;
END_VAR
VAR CONSTANT
	spoolSpacing : TIME := T#100MS;
	
	numTotalConveyors : INT := 38;
	
	numCellConveyors : INT := 20;
	
	numReceiverConveyors : INT := 6;
	numOutputConveyors : INT := 12;
END_VAR
(*
this module contains all conveyors to be distributed to subareas as needed
by not tying conveyors to any particular subarea, any subarea will have some access to any conveyor
*)

fillCellConveyors();
fillReceiverConveyors();
fillOutputConveyors();

computeCellLinks();

spoolTimer(IN:= , PT:= spoolSpacing, Q=> , ET=> );
spoolTimer.IN := TRUE;

IF
	( //conveyor requests motion
		cellConveyors[i]^.requestedMode = ConveyorMode.FORWARD OR 
		cellConveyors[i]^.requestedMode = ConveyorMode.BACKWARD
	) AND
	cellConveyors[i]^.requestedMode <> cellConveyors[i]^.trueMode AND //conveyor request differs from current operation
	spoolTimer.Q //ready to spool
THEN
	//spool up conveyor
	i := (i + 1) MOD (numCellConveyors + 1) + 1;
	spoolTimer.IN := FALSE;
END_IF

METHOD PRIVATE computeCellLinks : BOOL
VAR
	i : DINT;
	j : DINT;
	
	linkStart : DINT := -1;
	linkEnd : DINT := -1;
	
	priorityInLink : ConveyorMode;
END_VAR
(*
link interation method 
will correctly set all operations every cycle
*)
FOR i:=1 TO numCellConveyors BY 1 DO
	IF cellConveyors[i]^.IsOccupied THEN
		
		IF linkStart = -1 THEN
			linkStart := i;
		END_IF
		
		priorityInLink := MAX(priorityInLink, cellConveyors[i]^.requestedMode);
		linkEnd := i;
		
	ELSIF linkStart <> -1 AND linkEnd <> -1 THEN //set all conveyor operations to priorityInLink
		linkEnd := i-1;
		
		FOR j:=linkStart TO linkEnd BY 1 DO
			cellConveyors[j]^.setMode(priorityInLink);
		END_FOR
		
		linkStart := -1;
		linkEnd := -1;
		priorityInLink := ConveyorMode.IDLE;
		
		CONTINUE;
	END_IF
	
END_FOR


//final link
IF linkStart > -1 AND linkEnd > -1 THEN
	FOR j:=linkStart TO linkEnd BY 1 DO
		cellConveyors[j]^.setMode(priorityInLink);
	END_FOR
END_IF
END_METHOD

METHOD PRIVATE fillCellConveyors : BOOL
{warning disable C0371}
cellConveyors[1] := ADR(A24_SC_C01);
cellConveyors[2] := ADR(A24_SC_C03);
cellConveyors[3] := ADR(A24_SC_C05);
cellConveyors[4] := ADR(A24_SC_C07);
cellConveyors[5] := ADR(A24_SC_C09);
cellConveyors[6] := ADR(A24_SC_C11);
cellConveyors[7] := ADR(A24_SC_C13);

cellConveyors[8] := ADR(A23_LSC_C14);

cellConveyors[9] := ADR(A22_SC_C15);
cellConveyors[10] := ADR(A22_LSC_C16);
cellConveyors[11] := ADR(A22_LSC_C17);

cellConveyors[12] := ADR(A21_SC_C18);
cellConveyors[13] := ADR(A21_LSC_C19);
cellConveyors[14] := ADR(A21_LSC_C20);
cellConveyors[15] := ADR(A21_LSC_C21);

cellConveyors[16] := ADR(A25_SC_C22);
cellConveyors[17] := ADR(A25_SC_C24);
cellConveyors[18] := ADR(A25_SC_C26);
cellConveyors[19] := ADR(A25_SC_C28);
cellConveyors[20] := ADR(A25_SC_C30);
END_METHOD

METHOD PRIVATE fillOutputConveyors : BOOL
VAR_INPUT
END_VAR
outputConveyors[1] := ADR(A25_LSC_C23);
outputConveyors[2] := ADR(A25_LSLCC_C25);
outputConveyors[3] := ADR(A25_LSLCC_C27);
outputConveyors[4] := ADR(A25_LSC_C29);
outputConveyors[5] := ADR(A25_SC_C31);
outputConveyors[6] := ADR(A25_SC_C32);
outputConveyors[7] := ADR(A25_SC_C33);
outputConveyors[8] := ADR(A25_SC_C34);
outputConveyors[9] := ADR(A25_SC_C35);
outputConveyors[10] := ADR(A25_SC_C36);
outputConveyors[11] := ADR(A25_SC_C37);
outputConveyors[12] := ADR(A25_SC_C38);
END_METHOD

METHOD PRIVATE fillReceiverConveyors : BOOL
VAR_INPUT
END_VAR
receiverConveyors[1] := ADR(A24_LRC_C02);
receiverConveyors[2] := ADR(A24_LRC_C04);
receiverConveyors[3] := ADR(A24_LRC_C06);
receiverConveyors[4] := ADR(A24_LRC_C08);
receiverConveyors[5] := ADR(A24_LRC_C10);
receiverConveyors[6] := ADR(A24_LRC_C12);
END_METHOD

END_PROGRAM

// ---- HARDWARE_DISTRUBUTION/A22.TcPOU
FUNCTION_BLOCK A22 EXTENDS GenericSubarea
VAR_IN_OUT
	sectionCC : CardboardEx;
END_VAR
VAR
	robot3, robot4 : RobotA22;
	
	benderA22Left : FoldingMachine;
	
	skidA22Left, skidA22Right : SkidMagazine;
	magazineA22Left, magazineA22Right : SkidMagazine;
	
	wrapperA22 : WrapMachine;
	
	centeringSliderA22 : ServoNC;
	
	horizontalDriveA22Left, horizontalDriveA22Right : ServoNC := (
		limitSensorDefaultState := TRUE);
		
	verticalDriveA22Left, verticalDriveA22Right : ClearLinkMC := (
		limitSensorDefaultState := TRUE, 
		homingDirectionOut := TRUE, //outwards (up)
		minPosition := (26*5 * 25.4),
		displacementPerRotation := 5,
		unitsPerPulse := 800); //800 counts = 1 rotation
		
	insertionA22Left, insertionA22Right : Insertion;

	pistonA22Bottom : SimplePiston;
	
	(*
	each insertion suction array has 3 pads
	[1] - top/bottom
	[2] - corner
	[3] - side
	*)
	suctionA22TopLeft : ARRAY[1..3] OF SuctionPad;
	suctionA22TopRight : ARRAY[1..3] OF SuctionPad;
	suctionA22BottomLeft : ARRAY[1..3] OF SuctionPad; 
	suctionA22BottomRight : ARRAY[1..3] OF SuctionPad;
	
	suctionA22Bottom : ARRAY[1..2] OF SuctionPad;
END_VAR
VAR //data arrays to be passed into material holder FBs - do not access directly
	skidHmiA22Left, skidHmiA22Right AT %M* : ARRAY[1...Cardboard.size-1] OF MaterialSlot;
	magazineHmiA22Left, magazineHmiA22Right AT %M* : ARRAY[1..CornerGuard.size-1] OF MaterialSlot;
END_VAR
VAR //other
	conveyorsCC : ARRAY[1..3] OF POINTER TO ConveyorSC;
END_VAR

SUPER^();

METHOD PROTECTED callHardware : BOOL
skidA22Left(slots := skidHmiA22Left);
skidA22Right(slots := skidHmiA22Right);
magazineA22Left(slots := magazineHmiA22Left);
magazineA22Right(slots := magazineHmiA22Right);

wrapperA22(extSafety := robot3.wrapSafetyIn AND robot4.wrapSafetyIn);

verticalDriveA22Left(
	bEnable:= TRUE, 
	pulse=> , 
	brakeRelease=> , 
	enable=> , 
	A=> , 
	B=> , 
	clear=> );
verticalDriveA22Right(
	bEnable:= TRUE, 
	pulse=> , 
	brakeRelease=> , 
	enable=> , 
	A=> , 
	B=> , 
	clear=> );

horizontalDriveA22Left(bEnable:= TRUE, ready=> , position=> , velocity=> );
horizontalDriveA22Right(bEnable:= TRUE, ready=> , position=> , velocity=> );

insertionA22Left(
	slider:= verticalDriveA22Left, 
	screw:= horizontalDriveA22Left, 
	contact=> , 
	active=> , 
	error=> , 
	home=> , 
	homingComplete=> , 
	sliderPos=> );
	
insertionA22Right(
	slider:= verticalDriveA22Right, 
	screw:= horizontalDriveA22Right, 
	contact=> , 
	active=> , 
	error=> , 
	home=> , 
	homingComplete=> , 
	sliderPos=> );
END_METHOD

METHOD PROTECTED runModules : BOOL
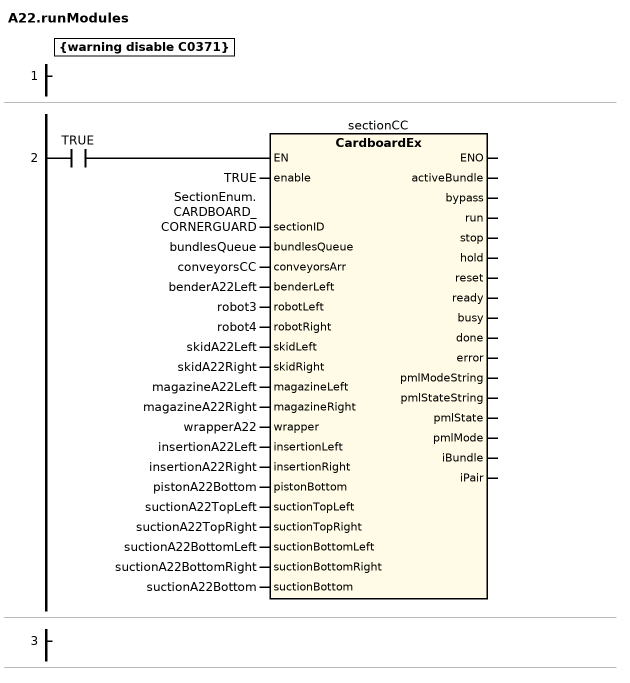
// NETWORK 1
// label: {warning disable C0371}

// NETWORK 2
sectionCC(
    enable := TRUE,
    sectionID := SectionEnum.CARDBOARD_CORNERGUARD,
    bundlesQueue := bundlesQueue,
    conveyorsArr := conveyorsCC,
    benderLeft := benderA22Left,
    robotLeft := robot3,
    robotRight := robot4,
    skidLeft := skidA22Left,
    skidRight := skidA22Right,
    magazineLeft := magazineA22Left,
    magazineRight := magazineA22Right,
    wrapper := wrapperA22,
    insertionLeft := insertionA22Left,
    insertionRight := insertionA22Right,
    pistonBottom := pistonA22Bottom,
    suctionTopLeft := suctionA22TopLeft,
    suctionTopRight := suctionA22TopRight,
    suctionBottomLeft := suctionA22BottomLeft,
    suctionBottomRight := suctionA22BottomRight,
    suctionBottom := suctionA22Bottom); // CardboardEx

// NETWORK 3
END_METHOD

METHOD PROTECTED setupHardware : BOOL
VAR
	iCornerGuardSlot : CornerGuard;
	iCardboardSlot : Cardboard;
	i : INT;
END_VAR
FOR iCornerGuardSlot:=1 TO WoodBunk.size-1 BY 1 DO //init wood bunk magazine slots
	magazineA22Left.setSlot(i := iCornerGuardSlot, material := TO_STRING(iCornerGuardSlot), error => );
	magazineA22Right.setSlot(i := iCornerGuardSlot, material := TO_STRING(iCornerGuardSlot), error => );
END_FOR

//--------------------------------------------------

FOR iCardboardSlot:=1 TO Chipboard.size-1 BY 1 DO //init chipboard skid slots
	skidA22Left.setSlot(i := iCardboardSlot, material := TO_STRING(iCardboardSlot), error => );
	skidA22Right.setSlot(i := iCardboardSlot, material := TO_STRING(iCardboardSlot), error => );
END_FOR

//--------------------------------------------------

FOR i:=1 TO CONSTS.maxQueue BY 1 DO //get corner guard magazine + cardboard skid availability from robot3 and robot4
	{warning disable C0195}
	skidA22Left.setOccupancy( i := i, occupancy := IntegerBitAccess(robot3.inputs[4], i-1) );
	skidA22Right.setOccupancy( i := i, occupancy := IntegerBitAccess(robot4.inputs[4], i-1) );

	magazineA22Left.setOccupancy( i := i, occupancy := IntegerBitAccess(robot4.inputs[3], i-1) );
	magazineA22Right.setOccupancy( i := i, occupancy := IntegerBitAccess(robot4.inputs[3], i-1) );
END_FOR

//--------------------------------------------------

conveyorsCC[1] := ADR(ConveyorSyncUnit.A22_SC_C15);
conveyorsCC[2] := ADR(ConveyorSyncUnit.A22_LSC_C16);
conveyorsCC[3] := ADR(ConveyorSyncUnit.A22_LSC_C17);
END_METHOD

END_FUNCTION_BLOCK

// ---- HARDWARE_DISTRUBUTION/A24.TcPOU
FUNCTION_BLOCK A24 EXTENDS GenericSubarea
VAR
	conveyors : ARRAY[1..6] OF POINTER TO Conveyor;
END_VAR
VAR
	step : (IDLE, RECEIVE, SEND, VACANT);
END_VAR

SUPER^();

CASE step OF
	IDLE:
		allConveyorsRequest(newRequest := ConveyorMode.IDLE);
		
		IF TRUE(*incoming bundle*) THEN
			step := RECEIVE;
		END_IF
		
	RECEIVE:
		allConveyorsRequest(newRequest := ConveyorMode.STOP);
		
		IF TRUE (*area 3 is done transferring*) THEN
			step := SEND;
		END_IF
		
	SEND:
		allConveyorsRequest(newRequest := ConveyorMode.FORWARD);
		
		IF allConveyorsVacant() THEN
			step := VACANT;
		END_IF
		
	VACANT:
		allConveyorsRequest(newRequest := ConveyorMode.IDLE);
		step := 0;
		
END_CASE

METHOD PROTECTED allConveyorsRequest : BOOL
VAR_INPUT
	newRequest : ConveyorMode;
END_VAR
VAR
	i : INT;
END_VAR
FOR i:=1 TO 6 BY 1 DO
	conveyors[i]^.setRequest(newRequest := newRequest);
END_FOR
END_METHOD

METHOD PROTECTED allConveyorsVacant : BOOL
VAR_INPUT
END_VAR
VAR
	i : INT;
END_VAR
FOR i:=1 TO 6 BY 1 DO
	IF conveyors[i]^.IsOccupied THEN
		RETURN;
	END_IF
END_FOR

allConveyorsVacant := TRUE;
END_METHOD

METHOD PROTECTED callHardware : BOOL
VAR_INPUT
END_VAR
END_METHOD

METHOD PROTECTED runModules : BOOL
VAR_INPUT
END_VAR
// NETWORK 1
END_METHOD

METHOD PROTECTED setupHardware : BOOL
VAR
	i : INT;
END_VAR
conveyors[1] := ADR(ConveyorSyncUnit.A24_LRC_C02);
conveyors[2] := ADR(ConveyorSyncUnit.A24_LRC_C04);
conveyors[3] := ADR(ConveyorSyncUnit.A24_LRC_C06);
conveyors[4] := ADR(ConveyorSyncUnit.A24_LRC_C08);
conveyors[5] := ADR(ConveyorSyncUnit.A24_LRC_C10);
conveyors[6] := ADR(ConveyorSyncUnit.A24_LRC_C12);
END_METHOD

END_FUNCTION_BLOCK

// ---- HARDWARE_DISTRUBUTION/A25.TcPOU
FUNCTION_BLOCK A25 EXTENDS GenericSubarea

SUPER^();

METHOD PROTECTED callHardware : BOOL
VAR_INPUT
END_VAR
END_METHOD

METHOD PROTECTED runModules : BOOL
VAR_INPUT
END_VAR
// NETWORK 1
END_METHOD

METHOD PROTECTED setupHardware : BOOL
VAR
	i : INT;
END_VAR
END_METHOD

END_FUNCTION_BLOCK

// ---- EventLogging/SqlDatabaseAccessor.TcPOU
FUNCTION_BLOCK SqlDatabaseAccessor IMPLEMENTS EventLogger //database logging, may be replaced with inbuilt eventlogger
VAR
	completedBundles : REFERENCE TO PtrQueue;
	
	events : IntQueue := (entrySize := 4); //local events queue
	
	fbSQLCommand : FB_SQLCommandEvt(sNetID := '', tTimeout := T#5S);
	fbSQLDatabase : FB_SQLDatabaseEvt (sNetID := '', tTimeout := T#5S);
	fbSQLResult: FB_SQLResultEvt(sNetID:='', tTimeout:=T#5S);
	
	queryOpening : STRING(1000) := 'INSERT INTO EventLog(Timestamp, Machine, Event, Type) VALUES(';
	fullQuery : STRING(1000);
	
	//for timestamps
	ntSystemTime : NT_GetTime;
    timeAsStruct : TIMESTRUCT;
	
	exeIn : ARRAY[0..2] OF STRING(1000);
	
	//iterators
	i : INT := 0;
	
	//step switch
	step : (IDLE,
			CONNECT_TO_DB, CREATE_CMD, INSERT_CMD, CLOSE_CONNECTION, 
			CONNECT_TO_LOCAL_DB, CREATE_LOCAL_CMD, INSERT_LOCAL_CMD, CLOSE_LOCAL_CONNECTION,
			ERROR);
END_VAR

CASE step OF //1-4 for local DB, 11-14 for plant DB
	//local EventLog DB should store all events for diagnosis
	IDLE:
		IF NOT events.isEmpty() THEN
			step := CONNECT_TO_DB;
		END_IF
		
	CONNECT_TO_DB: //open connection to local EventLog DB
		IF connectToDb() THEN
			step := 1;
		END_IF
		
	CREATE_CMD: //create command
		IF createCommand() THEN
			step := 2;
		END_IF
		
	INSERT_CMD: //insert command
		//timestamp, event, machine, type
		//ntSystemTime(NETID := , START := TRUE, TMOUT := DEFAULT_ADS_TIMEOUT, BUSY => , ERR =>, ERRID =>, TIMESTR => timeAsStruct);
		
		fullQuery := CONCAT(queryOpening, '$''); //timestamp
		fullQuery := CONCAT(fullQuery, TimestructToString(GVL.bundleOut.timeDone));
		fullQuery := CONCAT(fullQuery, '$', ');
		
		exeIn[0] := CONCAT(queryOpening, '$''); //timestamp
		exeIn[0] := CONCAT(fullQuery, TimestructToString(timeAsStruct));
		exeIn[0] := CONCAT(fullQuery, '$', ');
		
		CASE events.get(i:=0) OF //event
			(*EventsEnum.BUNDLE_SENT:
				exeIn[1] := CONCAT(exeIn[1], '$'Bundle Sent (');
				exeIn[1] := CONCAT(exeIn[1], GVL.bundleOut^.id);
				exeIn[1] := CONCAT(exeIn[1], ')$'');*)
			EventsEnum.BACKLOG:
				exeIn[1] := CONCAT(exeIn[1], '$'Backlog$'');
			EventsEnum.MACHINE_FAILURE: //and other specific events to be logged
				exeIn[1] := CONCAT(exeIn[1], '$'Machine Failure$'');
			EventsEnum.DELAY:
				exeIn[1] := CONCAT(exeIn[1], '$'Delay (');
				exeIn[1] := CONCAT(exeIn[1], GVL.bundleOut.id);
				exeIn[1] := CONCAT(exeIn[1], ')$'');
			EventsEnum.BUNDLE_LATE_RECEIVED:
				exeIn[1] := CONCAT(exeIn[1], '$'Late Arrival (');
				exeIn[1] := CONCAT(exeIn[1], GVL.bundleOut.id);
				exeIn[1] := CONCAT(exeIn[1], ')$'');
			EventsEnum.BUNDLE_EARLY_RECEIVED:
				exeIn[1] := CONCAT(exeIn[1], '$'Early Arrival (');
				exeIn[1] := CONCAT(exeIn[1], GVL.bundleOut.id);
				exeIn[1] := CONCAT(exeIn[1], ')$'');
			ELSE
				exeIn[1] := CONCAT(exeIn[1], '$'Other/Unknown$'');
		END_CASE
		
		exeIn[2] := CONCAT(exeIn[2], '$'Area 2$')'); //machine
		
		//ADSLOGSTR(msgCtrlMask := ADSLOG_MSGTYPE_ERROR OR ADSLOG_MSGTYPE_MSGBOX, msgFmtStr := sCMD, strArg := strSFCErrorStep);
		
		FOR i:=0 TO 2 BY 1 DO
			fullQuery := CONCAT(fullQuery, exeIn[i]);
		END_FOR
		
		IF fbSQLCommand.Execute(ADR(fullQuery), SIZEOF(fullQuery)) THEN
			step := 3;
		END_IF
	
	//3: //send data to system EventLog DB via TCP client
		(*IF client.send(sAction := 'log event', sData := sCMD) THEN
			step := 4;
		END_IF*)
		
	CLOSE_CONNECTION: //close connection
		events.poll();
		IF fbSQLDatabase.Disconnect() THEN
			step := 100;
		END_IF
	
	//system EventLog DB should only store simplified events
	(*100:
		IF NOT events.isEmpty() THEN
			IF fbSQLDatabase.Connect(5) THEN
				step := 11;
			END_IF
		END_IF
	
	101:
		IF fbSQLDatabase.CreateCmd(ADR(fbSQLCommand)) THEN
			step := 12;
		END_IF
	
	102:
		sCMD := CONCAT(CMD_0, '$''); //timestamp
		sCMD := CONCAT(sCMD, helper.timestructToString(timeAsStruct));
		sCMD := CONCAT(sCMD, '$', ');
		
		CASE events.get(i := 0) OF //event
			EventsEnum.BUNDLE_SENT:
				sCMD := CONCAT(sCMD, '$'Bundle Sent (');
				sCMD := CONCAT(sCMD, GVL.bundleOut^.id);
				sCMD := CONCAT(sCMD, ')$'');
			EventsEnum.BACKLOG:
				sCMD := CONCAT(sCMD, '$'Backlog$'');
			EventsEnum.MACHINE_FAILURE:
				sCMD := CONCAT(sCMD, '$'Machine Failure$'');
			EventsEnum.DELAY:
				sCMD := CONCAT(sCMD, '$'Delay (');
				sCMD := CONCAT(sCMD, GVL.bundleOut^.id);
				sCMD := CONCAT(sCMD, ')$'');
			EventsEnum.BUNDLE_LATE_RECEIVED:
				sCMD := CONCAT(sCMD, '$'Late Arrival (');
				sCMD := CONCAT(sCMD, GVL.bundleOut^.id);
				sCMD := CONCAT(sCMD, ')$'');
			EventsEnum.BUNDLE_EARLY_RECEIVED:
				sCMD := CONCAT(sCMD, '$'Early Arrival (');
				sCMD := CONCAT(sCMD, GVL.bundleOut^.id);
				sCMD := CONCAT(sCMD, ')$'');
			ELSE
				sCMD := CONCAT(sCMD, '$'Other/Unknown$'');
		END_CASE
		
		sCMD := CONCAT(sCMD, '$'Area 2$')'); //machine
		
		ADSLOGSTR(msgCtrlMask := ADSLOG_MSGTYPE_ERROR OR ADSLOG_MSGTYPE_MSGBOX, msgFmtStr := sCMD, strArg := strSFCErrorStep);
		
		IF fbSQLCommand.Execute(ADR(sCMD), SIZEOF(sCMD)) THEN
			step := 3;
		END_IF
	
	103:
		
	104:*)
		
		
END_CASE

METHOD connectToDb : BOOL
VAR_INPUT
END_VAR
IF fbSQLDatabase.Connect(1) THEN
	connectToDb := TRUE;
	RETURN;
END_IF
END_METHOD

METHOD createCommand : BOOL
VAR_INPUT
END_VAR
IF fbSQLDatabase.CreateCmd(ADR(fbSQLCommand)) THEN
	createCommand := TRUE;
	RETURN;
END_IF
END_METHOD

METHOD insertCommand : BOOL
VAR_INPUT
END_VAR
VAR
	tempPtr : POINTER TO Bundle;
END_VAR
//for bundle completion events use bundle.timeDone, otherwise use system time
IF events.get(i:=0) = EventsEnum.BUNDLE_COMPLETE THEN
	tempPtr := completedBundles.poll();
	timeAsStruct := tempPtr^.timeDone;
	__DELETE(tempPtr);
ELSE
	ntSystemTime(NETID := , START := TRUE, TMOUT := DEFAULT_ADS_TIMEOUT, BUSY => , ERR =>, ERRID =>, TIMESTR => timeAsStruct);
END_IF

fullQuery := CONCAT(queryOpening, '$''); //timestamp
fullQuery := CONCAT(fullQuery, TimestructToString(GVL.bundleOut.timeDone));
fullQuery := CONCAT(fullQuery, '$', ');

exeIn[0] := CONCAT(queryOpening, '$''); //timestamp
exeIn[0] := CONCAT(fullQuery, TimestructToString(timeAsStruct));
exeIn[0] := CONCAT(fullQuery, '$', ');

CASE events.get(i:=0) OF //event
	(*EventsEnum.BUNDLE_SENT:
		exeIn[1] := CONCAT(exeIn[1], '$'Bundle Sent (');
		exeIn[1] := CONCAT(exeIn[1], GVL.bundleOut^.id);
		exeIn[1] := CONCAT(exeIn[1], ')$'');*)
	EventsEnum.BACKLOG:
		exeIn[1] := CONCAT(exeIn[1], '$'Backlog$'');
	EventsEnum.MACHINE_FAILURE: //and other specific events to be logged
		exeIn[1] := CONCAT(exeIn[1], '$'Machine Failure$'');
	EventsEnum.DELAY:
		exeIn[1] := CONCAT(exeIn[1], '$'Delay (');
		exeIn[1] := CONCAT(exeIn[1], GVL.bundleOut.id);
		exeIn[1] := CONCAT(exeIn[1], ')$'');
	EventsEnum.BUNDLE_LATE_RECEIVED:
		exeIn[1] := CONCAT(exeIn[1], '$'Late Arrival (');
		exeIn[1] := CONCAT(exeIn[1], GVL.bundleOut.id);
		exeIn[1] := CONCAT(exeIn[1], ')$'');
	EventsEnum.BUNDLE_EARLY_RECEIVED:
		exeIn[1] := CONCAT(exeIn[1], '$'Early Arrival (');
		exeIn[1] := CONCAT(exeIn[1], GVL.bundleOut.id);
		exeIn[1] := CONCAT(exeIn[1], ')$'');
	ELSE
		exeIn[1] := CONCAT(exeIn[1], '$'Other/Unknown$'');
END_CASE

exeIn[2] := CONCAT(exeIn[2], '$'Area 2$')'); //machine

//ADSLOGSTR(msgCtrlMask := ADSLOG_MSGTYPE_ERROR OR ADSLOG_MSGTYPE_MSGBOX, msgFmtStr := sCMD, strArg := strSFCErrorStep);
END_METHOD

METHOD logEvent : BOOL
VAR_INPUT
END_VAR
END_METHOD

METHOD queueEvent : BOOL
VAR_INPUT
	event : INT;
END_VAR
events.push(event);
END_METHOD

END_FUNCTION_BLOCK

// ---- DUTs/Containers/PtrQueue.TcPOU
FUNCTION_BLOCK PtrQueue EXTENDS Queue //stores pointers to bundles, not the bundles themselves
VAR_INPUT
	
END_VAR
VAR
	elements : FB_BA_DynamicArray := (uiEntrySize := SIZEOF(PVOID), uiMinExpCount := CONSTS.initArraySize);
	//length : USINT := 0;
END_VAR

METHOD get : PVOID;
VAR_INPUT
	i : UINT;
END_VAR
elements.GetEntry(diIndex := i, pResultEntry := ADR(get));
END_METHOD

METHOD isEmpty : BOOL
VAR_INPUT
END_VAR
isEmpty := (elements.diCount = 0);
END_METHOD

METHOD poll : PVOID;
VAR_INST
	i : UINT;
END_VAR
poll := get(i := 0);
elements.RemoveEntry(diIndex := 0);
//length := length - 1;
END_METHOD

METHOD push : BOOL
VAR_INPUT
	value : PVOID;
END_VAR
elements.AddEntryPtr(pEntry := value);
//length := length + 1;
push := TRUE;
END_METHOD

METHOD size : DINT
VAR_INPUT
END_VAR
size := elements.diCount;
END_METHOD

END_FUNCTION_BLOCK

// ---- POUs/TypeSizeCheck.TcPOU
PROGRAM TypeSizeCheck
VAR
	bundleSize : ULINT;
	adsDataSize : ULINT;
	tcpDataSize : ULINT;
	allSectionSize : ULINT;
END_VAR

bundleSize := SIZEOF(Bundle);
adsDataSize := SIZEOF(AdsData);
tcpDataSize := SIZEOF(TcpData);

allSectionSize := SIZEOF(WoodBunkEx) + SIZEOF(ChipboardEx) + SIZEOF(SpacerRecollectionUnit);

END_PROGRAM

// ---- COMs/Comms_ADS/AdsTcpUnitEx.TcPOU
FUNCTION_BLOCK AdsTcpUnitEx
VAR_INPUT
	setMode : (SEND, QUEUE);
END_VAR
VAR_OUTPUT
	bBusy : BOOL;
	error : BOOL;
	errorID : UDINT;
END_VAR
VAR
	socketsArr : ARRAY[1..numSockets] OF POINTER TO AdsSocket; //use this to find a socket
	
	//declare all sockets here
	AREA_2 : AdsSocket := (PrgName := TO_STRING(AreaEnum.AREA_2), AmsNetId := '192.168.101.188.1.1', AmsPort := 851);
	AREA_3 : AdsSocket := (PrgName := TO_STRING(AreaEnum.AREA_3), AmsNetId := '3.0.131.216.1.1', AmsPort := 851); //placeholder NetId
END_VAR
VAR
	socket : REFERENCE TO AdsSocket;
	
	messageQueue : AdsMessageQueue;
	nextMessage : AdsMessage;
	
	mode : (SEND, QUEUE);
END_VAR
VAR CONSTANT
	numSockets : INT := 2;
END_VAR

(*
	this TCP-style ADS communication module provides the option to dynamically generate ADS messages into a queue
		due to the significant stack memory requirements, the QUEUE model can only be used on systems with adjustable stack
		using QUEUE mode on panel PCs (CP66xx) or other mini controllers can freeze the system
		
	QUEUE mode:
		when a message is polled, a socket with the same recipient name is identified
			if the identified socket is ready to send, then the message is passed to the socket
			otherwise, the message is placed back into the queue
		if no socket with a matching name can be identified, then the message is discarded
		
	SEND mode:
		if a socket matching the recipient name is identified and it is not busy or in error state, then the message is passed
		
	sendMessage() specifies a recipient name and data contents, then checks the mode to determine how to handle the message
*)

fillSocketsArr();

IF messageQueue.isEmpty() THEN
	mode := setMode;
END_IF

blocks();

IF mode = QUEUE THEN
	pollAndSend();	
END_IF

METHOD PRIVATE blocks : BOOL
VAR_INPUT
END_VAR
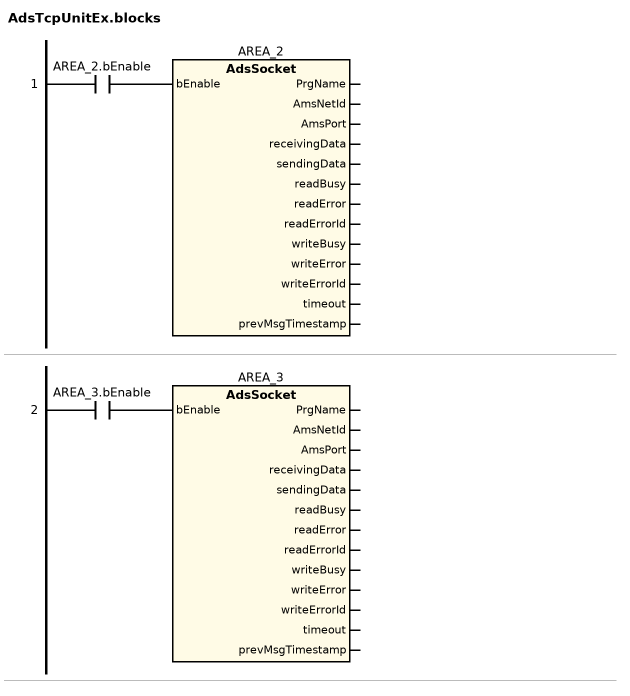
// NETWORK 1
AREA_2(bEnable := AREA_2.bEnable); // AdsSocket

// NETWORK 2
AREA_3(bEnable := AREA_3.bEnable); // AdsSocket
END_METHOD

METHOD fetchData : BOOL
VAR_INPUT
	senderName : STRING;
END_VAR
VAR_OUTPUT
	data : AdsData;
END_VAR
VAR
	i : INT;
END_VAR
FOR i:=1 TO numSockets BY 1 DO
	
	IF socketsArr[i]^.PrgName = senderName THEN
		fetchData := TRUE;
		data := socketsArr[i]^.receivingData;
		RETURN;
	END_IF
	
END_FOR
END_METHOD

METHOD PRIVATE fillSocketsArr : BOOL
VAR_INPUT
END_VAR
socketsArr[1] := ADR(AREA_2);
socketsArr[2] := ADR(AREA_3);
END_METHOD

METHOD PRIVATE findSocket : REFERENCE TO AdsSocket
VAR_INPUT
	recipient : STRING;
END_VAR
VAR
	i : INT;
END_VAR
FOR i:=1 TO numSockets BY 1 DO
	IF socketsArr[i] <> 0 AND_THEN socketsArr[i]^.PrgName = recipient THEN
		findSocket REF= socketsArr[i]^;
		RETURN;
	END_IF
END_FOR
END_METHOD

METHOD PRIVATE pollAndSend : BOOL
VAR_INPUT
END_VAR
nextMessage := messageQueue.poll(getSize => );
socket REF= findSocket(recipient := nextMessage.recipient);

IF __ISVALIDREF(socket) THEN
	
	IF NOT socket.writeBusy AND NOT socket.writeError AND socket.writeReady THEN
		socket.send(data := nextMessage.contents);
	ELSE //if socket is busy or has ERROR state, then message is returned to the end of the line
		messageQueue.push(value := nextMessage);
	END_IF
	
END_IF
END_METHOD

METHOD sendMessage : BOOL
VAR_INPUT
	recipient : STRING;
	data : REFERENCE TO AdsData;
END_VAR
VAR
	newMessage : AdsMessage;
END_VAR
CASE mode OF
	SEND:
		socket REF= findSocket(recipient := recipient);
		IF
			__ISVALIDREF(socket) AND_THEN
			NOT socket.writeBusy AND NOT socket.writeError
		THEN
			socket.send(data := data);
			sendMessage := TRUE;
		END_IF
	
	QUEUE:
		IF recipient <> '' THEN
			newMessage.recipient := recipient;
			newMessage.contents := data;
			
			sendMessage := messageQueue.push(newMessage);
		END_IF
	
END_CASE
END_METHOD

END_FUNCTION_BLOCK

// ---- COMs/Comms_ADS/AdsSocket.TcPOU
FUNCTION_BLOCK AdsSocket
VAR_INPUT
	bEnable : BOOL;
END_VAR
VAR_OUTPUT
	PrgName : STRING; //descriptive string for the name of the running program
	AmsNetId : T_AmsNetId; //this must be assigned even if it is used for local communication - otherwise socket is not considered valid
	AmsPort : T_AmsPort; //for now, use ADS port 851 for communication
END_VAR
VAR_OUTPUT
	receivingData : AdsData;
	sendingData : AdsData;
	
	readBusy : BOOL;
	readError : BOOL;
	readErrorId : UDINT;
	
	writeBusy : BOOL;
	writeError : BOOL;
	writeErrorId : UDINT;
	
	writeReady : BOOL;
	
	timeout : BOOL;
	prevMsgTimestamp : TIMESTRUCT;
END_VAR
VAR	
	targetSocket : STRING := CONCAT('COM.adsMajorNetwork.', localPrgName); //write into the recipient's allocated socket for this system
	adsWriteSymbol : FB_WriteAdsSymByName;
	adsReadSymbol : FB_ReadAdsSymByName;
END_VAR
VAR	
	toggleBit : BOOL; //remote system toggles this bit - use as heartbeat input
	sendingBit : BOOL; //this system toggles this bit - write to remote system's toggleBit
	
	heartbeat : Watchdog;
	writeDelayTimer : TON;
	
	flagWriter : FB_WriteAdsSymByName;
	nameWriter : FB_WriteAdsSymByName;
	netIdWriter : FB_WriteAdsSymByName;
	portWriter : FB_WriteAdsSymByName;
	
	writeSync : BOOL := FALSE;
END_VAR
VAR_STAT
	fbGetLocalAmsNetId : FB_GetLocalAmsNetId;
	
	localPrgName : STRING := TO_STRING(AreaEnum.AREA_2);
	localAmsNetId : T_AmsNetId := '';
	localAmsPort : T_AmsPort := 851;
	
	writeSpacing : TIME := T#200MS;
END_VAR
(*
TCP-style ADS connection that only writes to a buffer in the recipient's AdsTcpUnit module
*)

writeDelayTimer(IN:= NOT writeBusy, PT:= writeSpacing, Q=> writeReady, ET=> );

targetSocket := CONCAT('COM.adsMajorNetwork.', localPrgName);

flagSequence();

IF //do not use this socket if invalid
	NOT bEnable OR
	NOT IsValid
THEN
	RETURN;
END_IF

setup();

(*
if timeout, stop all read/write
if data has no contents, do not send
*)
adsReadSymbol.bRead := NOT timeout AND NOT adsReadSymbol.bRead AND adsReadSymbol.sVarName <> '';
adsWriteSymbol.bWrite := 
	NOT timeout AND
	NOT BufferIsEmpty(sendingData.binaryData) AND 
	NOT adsWriteSymbol.bWrite;

blocks();

(*
IF timeout THEN //stop data read/write attempts
	adsWriteSymbol.bWrite := FALSE;
	adsReadSymbol.bRead := FALSE;
	
ELSE //only writes if data has contents, otherwise remains false
	adsWriteSymbol.bWrite := NOT BufferIsEmpty(sendingData.binaryData) AND NOT adsWriteSymbol.bWrite;
END_IF
*)

METHOD PRIVATE blocks : BOOL
VAR_INPUT
END_VAR
adsReadSymbol(
	bRead:= , 
	sNetId:= AmsNetId, 
	nPort:= AmsPort, 
	sVarName:= , 
	nDestAddr:= , 
	nLen:= , 
	tTimeout:= , 
	eComMode:= , 
	bClearOnError:= , 
	bBusy=> readBusy, 
	bError=> readError, 
	nErrorId=> readErrorId);
	
adsWriteSymbol(
	bWrite:= , 
	sNetId:= AmsNetId, 
	nPort:= AmsPort, 
	sVarName:= CONCAT(targetSocket, '.receivingData'), 
	nSrcAddr:= ADR(sendingData), 
	nLen:= SIZEOF(sendingData), 
	tTimeout:= , 
	eComMode:= eAdsComModeSecureCom, 
	bBusy=> writeBusy, 
	bError=> writeError, 
	nErrorId=> writeErrorId);
	
IF NOT adsWriteSymbol.bBusy THEN
	MEMSET(ADR(sendingData), 0, SIZEOF(sendingData));
END_IF
END_METHOD

METHOD PRIVATE flagSequence : BOOL
VAR_INPUT
END_VAR
heartbeat(
	enable:= TRUE, 
	toggleBit:= toggleBit, 
	timeoutWidth:= DEFAULT_ADS_TIMEOUT, 
	timeout=> timeout);

prevMsgTimestamp := heartbeat.prevMsgTimestamp;

IF NOT flagWriter.bBusy THEN
	sendingBit := NOT sendingBit;
END_IF
END_METHOD

{attribute 'monitoring' := 'call'}
PROPERTY IsValid : BOOL
GET
IsValid := 
	PrgName <> '' AND
	AmsNetId <> '' AND
	AmsPort <> 0;
END_GET
END_PROPERTY

METHOD send : BOOL
VAR_INPUT
	data : REFERENCE TO AdsData;
END_VAR
sendingData := data;
END_METHOD

METHOD PRIVATE setup : BOOL
VAR_INST
	name : STRING;
END_VAR
fbGetLocalAmsNetId(
	bExecute:= (localAmsNetId = '' OR localAmsNetId = '0.0.0.0.0.0') AND NOT fbGetLocalAmsNetId.bExecute, 
	tTimeOut:= , 
	bBusy=> , 
	bError=> , 
	nErrId=> , 
	AddrString=> localAmsNetId, 
	AddrBytes=> );

writeSync := NOT writeSync;

nameWriter(
	bWrite:= writeSync, 
	sNetId:= AmsNetId, 
	nPort:= AmsPort, 
	sVarName:= CONCAT(targetSocket, '.PrgName'), 
	nSrcAddr:= ADR(localPrgName), 
	nLen:= SIZEOF(localPrgName), 
	tTimeout:= , 
	eComMode:= , 
	bBusy=> , 
	bError=> , 
	nErrorId=> );
	
netIdWriter(
	bWrite:= writeSync, 
	sNetId:= AmsNetId, 
	nPort:= AmsPort, 
	sVarName:= CONCAT(targetSocket, '.AmsNetId'), 
	nSrcAddr:= ADR(localAmsNetId), 
	nLen:= SIZEOF(localAmsNetId), 
	tTimeout:= , 
	eComMode:= , 
	bBusy=> , 
	bError=> , 
	nErrorId=> );
	
portWriter(
	bWrite:= writeSync, 
	sNetId:= AmsNetId, 
	nPort:= AmsPort, 
	sVarName:= CONCAT(targetSocket, '.AmsPort'), 
	nSrcAddr:= ADR(localAmsPort), 
	nLen:= SIZEOF(localAmsPort), 
	tTimeout:= , 
	eComMode:= , 
	bBusy=> , 
	bError=> , 
	nErrorId=> );
	
flagWriter(
	bWrite:= writeSync, 
	sNetId:= AmsNetId, 
	nPort:= AmsPort, 
	sVarName:= CONCAT(targetSocket, '.toggleBit'), 
	nSrcAddr:= ADR(sendingBit), 
	nLen:= SIZEOF(sendingBit), 
	tTimeout:= , 
	eComMode:= , 
	bBusy=> , 
	bError=> , 
	nErrorId=> );
END_METHOD

END_FUNCTION_BLOCK

// ---- COMs/Comms_ADS/AdsMessageQueue.TcPOU
{attribute 'call_after_init'}
FUNCTION_BLOCK AdsMessageQueue
VAR
	//elements : FB_BA_DynamicArray := (uiEntrySize := SIZEOF(POINTER TO AdsMessage), uiMinExpCount := 4);
	
	elements : FB_BA_StaticArray := (uiEntrySize := SIZEOF(POINTER TO AdsMessage), pExtMemory := ADR(arr), uiExtMemorySize := SIZEOF(arr));
	arr : ARRAY[0..99] OF POINTER TO AdsMessage;
	
	length : INT := 0;
	entrySize : UDINT;
END_VAR
VAR_STAT CONSTANT
	maxElements : INT := 100;
END_VAR
(*
this container stores dynamically generated AdsData Structs
AdsData to be added are passed by reference, then this function block allocates a structure to be stored
AdsData are get() by reference and poll() by value
*)

METHOD clear : BOOL
VAR
	i : INT;
	tempRef : REFERENCE TO AdsMessage;
	tempAdr : POINTER TO AdsMessage;
END_VAR
FOR i:=0 TO length-1 BY 1 DO
	tempRef := get(index := i, getSize => );
	tempAdr := ADR(tempRef);
	IF tempAdr <> 0 THEN
		__DELETE(tempAdr);
	END_IF
	
END_FOR

elements.Reset();
length := 0;
END_METHOD

